// TIA Portal project "Tartak_Projekt" (V14)

(* hardware
DEVICE "S7-1200 station_1"  S7-1200 Station
   slot 0: "Rack_0"  S7-1200 Rack  Rack  V1.0
   slot 1: "PLC_1"  CPU 1214C DC/DC/DC  6ES7 214-1AG31-0XB0  V3.0
      slot 3: "AQ 1x12BIT_1"  AQ1 signal board  6ES7 232-4HA30-0XB0  V1.0
   slot 2: "DI 16/DQ 16x24VDC_1"  SM 1223 DI16/DQ16 x 24VDC  6ES7 223-1BL30-0XB0  V1.0
DEVICE "HMI_2"  TP700 Comfort
   slot 0: "TP700 Comfort"  TP700 Comfort  6AV2 124-0GC01-0AX0  14.0.1.0
   slot 1: "HMI_RT_2"  TP700 Comfort  6AV2 124-0GC01-0AX0  14.0.1.0
   slot 5: "HMI_1.IE_CP_1"  PROFINET Interface  14.0.1.0
      slot 1: "PROFINET Interface_1"  PROFINET Interface
         slot 1: "Port_1"  Port
         slot 2: "Port_2"  Port
   slot 7: "HMI_1.MPI/DP_CP_1"  MPI/DP Interface  14.0.1.0
*)

// ===== PLC "PLC_1"  CPU 1214C DC/DC/DC =====

VAR_GLOBAL   // PLC tag table "Non Default tag table2"
   "Tag_1" AT %M100.0 : Bool;
   "Tag_2" AT %M100.1 : Bool;
   "Tag_3" AT %M100.2 : Bool;
   "Tag_4" AT %M100.3 : Bool;
   "Tag_5" AT %M100.4 : Bool;
   "Tag_6" AT %M100.5 : Bool;
   "Tag_7" AT %M1000.0 : Bool;
   "Tag_8" AT %M1000.1 : Bool;
   "Tag_9" AT %M1000.2 : Bool;
   "Tag_10" AT %M1000.3 : Bool;
   "Tag_11" AT %M1000.4 : Bool;
   "Tag_12" AT %M1000.5 : Bool;
   "Tag_13" AT %M1000.6 : Bool;
   "Tag_14" AT %M1000.7 : Bool;
   "Tag_15" AT %M1001.0 : Bool;
   "Tag_16" AT %M1001.1 : Bool;
   "Tag_17" AT %M1001.2 : Bool;
   "Tag_18" AT %M1001.3 : Bool;
   "Tag_19" AT %M1002.0 : Bool;
   "Tag_20" AT %M1002.1 : Bool;
   "Tag_21" AT %M2001.0 : Bool;
END_VAR

VAR_GLOBAL   // PLC tag table "Default tag table"
   "polozenie_dluga" AT %I8.0 : Bool;
   "polozenie_srednia" AT %I8.1 : Bool;
   "polozenie_krotka" AT %I8.2 : Bool;
   "polozenie_zsyp_1" AT %I8.3 : Bool;
   "polozenie_zsyp_2" AT %I8.4 : Bool;
   "polozenie_zsyp_3" AT %I8.5 : Bool;
   "P1" AT %Q4.0 : Bool;   // Przepychacz belek krótkich
   "P2" AT %Q4.1 : Bool;   // Przepychacz belek średnich
   "P3" AT %Q4.2 : Bool;   // Przepychacz belek długich
   "otwarcie_zsyp_1" AT %Q4.3 : Bool;
   "otwarcie_zsyp_2" AT %Q4.4 : Bool;
   "otwarcie_zsyp_3" AT %Q4.5 : Bool;
   "napelnienie_zsyp_1" AT %I8.6 : Bool;
   "napelnienie_zsyp_2" AT %I8.7 : Bool;
   "napelnienie_zsyp_3" AT %I9.0 : Bool;
   "pozycja_wagnik_zsyp_1" AT %I9.7 : Bool;
   "pozycja_wagonik_zsyp_2" AT %I1.0 : Bool;
   "pozycja_wagonik_zsyp_3" AT %I1.1 : Bool;
   "ruch_wagonika" AT %Q4.6 : Bool;
   "zwrotnica_bit_0" AT %Q4.7 : Bool;
   "zwrotnica_bit_1" AT %Q5.0 : Bool;
   "bocznica_dolna_0" AT %I9.1 : Bool;
   "bocznica_dolna_1" AT %I9.2 : Bool;
   "bocznica_srodkowa_0" AT %I9.3 : Bool;
   "bocznica_srodkowa_1" AT %I9.4 : Bool;
   "bocznica_gorna_0" AT %I9.5 : Bool;
   "bocznica_gorna_1" AT %I9.6 : Bool;
   "sygnalizator_gora" AT %Q5.1 : Bool;
   "sygnalizator_srodek" AT %Q5.2 : Bool;
   "sygnalizator_dol" AT %Q5.3 : Bool;
   "Clock_Byte" AT %MB0 : Byte;
   "Clock_10Hz" AT %M0.0 : Bool;
   "Clock_5Hz" AT %M0.1 : Bool;
   "Clock_2.5Hz" AT %M0.2 : Bool;
   "Clock_2Hz" AT %M0.3 : Bool;
   "Clock_1.25Hz" AT %M0.4 : Bool;
   "Clock_1Hz" AT %M0.5 : Bool;
   "Clock_0.625Hz" AT %M0.6 : Bool;
   "Clock_0.5Hz" AT %M0.7 : Bool;
   "alarmy" AT %MW10 : Int;
   "odbiorca" AT %M12.0 : Bool;
   "zsyp_1_krotka" AT %M50.0 : Bool;
   "zsyp_1_srednia" AT %M50.1 : Bool;
   "zsyp_1_dluga" AT %M50.2 : Bool;
   "zsyp_2_krotka" AT %M50.3 : Bool;
   "zsyp_2_srednia" AT %M50.4 : Bool;
   "zsyp_2_dluga" AT %M50.5 : Bool;
   "zsyp_3_krotka" AT %M50.6 : Bool;
   "zsyp_3_srednia" AT %M50.7 : Bool;
   "zsyp_3_dluga" AT %M51.0 : Bool;
END_VAR

VAR_GLOBAL CONSTANT   // PLC tag table "Default tag table"
   "None" : Pip := 65535;
   "Automatic update" : Pip := 0;
   "PIP 1" : Pip := 1;
   "PIP 2" : Pip := 2;
   "PIP 3" : Pip := 3;
   "PIP 4" : Pip := 4;
   "PIP OB Servo" : Pip := 32768;
   "Local~MC" : Hw_SubModule := 51;
   "Local~Common" : Hw_SubModule := 50;
   "Local~Device" : Hw_Device := 32;
   "Local~Configuration" : Hw_SubModule := 33;
   "Local~Exec" : Hw_SubModule := 52;
   "Local(1)" : Hw_SubModule := 49;
   "Local~PROFINET_interface_1(1)" : Hw_Interface := 64;
   "Local~PROFINET_interface_1~Port_1(1)" : Hw_Interface := 65;
   "Local~HSC_1(1)" : Hw_Hsc := 257;
   "Local~HSC_2(1)" : Hw_Hsc := 258;
   "Local~HSC_3(1)" : Hw_Hsc := 259;
   "Local~HSC_4(1)" : Hw_Hsc := 260;
   "Local~HSC_5(1)" : Hw_Hsc := 261;
   "Local~HSC_6(1)" : Hw_Hsc := 262;
   "Local~AI_2_1(1)" : Hw_SubModule := 263;
   "Local~DI_14_DQ_10_1(1)" : Hw_SubModule := 264;
   "Local~Pulse_1(1)" : Hw_Pwm := 265;
   "Local~Pulse_2(1)" : Hw_Pwm := 266;
   "Local~Pulse_3(1)" : Hw_Pwm := 267;
   "Local~Pulse_4(1)" : Hw_Pwm := 268;
   "OB_Main(1)" : OB_PCYCLE := 1;
END_VAR

DATA_BLOCK "DB_HMI"   // DB1
{ S7_Optimized_Access := 'TRUE' }
VERSION : 0.1
   VAR
      napelnienie_zsyp_krotki : Bool;
      napelnienie_zsyp_sredni : Bool;
      napelnienie_zsyp_dlugi : Bool;
      belka_krotka : Bool;
      belka_srednia : Bool;
      belka_dluga : Bool;
      status_ruchu_wagonika : Bool;
      oproznianie_zsyp_krotki : Bool;
      oproznianie_zsyp_sredni : Bool;
      oproznianie_zsyp_dlugi : Bool;
      ustawienie_zwrotnicy : Byte;
      zapelnienie_bocznicy_krotkiej : Byte;
      zapelnienie_bocznicy_sredniej : Byte;
      zapelnienie_bocznicy_dlugiej : Byte;
      sygnalizator_bocznica_krotka : Bool;
      sygnalizator_bocznica_srednia : Bool;
      sygnalizator_bocznica_dluga : Bool;
      wagonik_krotki : Bool;
      wagonik_sredni : Bool;
      wagonik_dlugi : Bool;
      odbiorca : Bool;
      zsyp_1_krotka : Bool;
      zsyp_1_srednia : Bool;
      zsyp_1_dluga : Bool;
      zsyp_2_krotka : Bool;
      zsyp_2_srednia : Bool;
      zsyp_2_dluga : Bool;
      zsyp_3_krotka : Bool;
      zsyp_3_srednia : Bool;
      zsyp_3_dluga : Bool;
   END_VAR
BEGIN
END_DATA_BLOCK

DATA_BLOCK "wykrywanie_belki_i_zrzucanie_DB"   // DB2
{ S7_Optimized_Access := 'TRUE' }
VERSION : 0.1
// stored: InstanceOfName wykrywanie_belki_i_zrzucanie
"wykrywanie_belki_i_zrzucanie"
BEGIN
END_DATA_BLOCK

DATA_BLOCK "poruszanie_wagonikiem_i_zsypywanie_drewna_DB"   // DB3
{ S7_Optimized_Access := 'TRUE' }
VERSION : 0.1
// stored: InstanceOfName poruszanie_wagonikiem_i_zsypywanie_drewna
"poruszanie_wagonikiem_i_zsypywanie_drewna"
BEGIN
END_DATA_BLOCK

DATA_BLOCK "wykrywanie_belki_i_zrzucanie_odbiorca_DB"   // DB6
{ S7_Optimized_Access := 'TRUE' }
VERSION : 0.1
// stored: InstanceOfName wykrywanie_belki_i_zrzucanie_odbiorca
"wykrywanie_belki_i_zrzucanie_odbiorca"
BEGIN
END_DATA_BLOCK

// folder: System blocks/Program resources

DATA_BLOCK "IEC_Timer_0_DB"   // DB4
{ S7_Optimized_Access := 'TRUE' }
AUTHOR : Simatic
FAMILY : IEC
NAME : IEC_TMR
VERSION : 1.0
// stored: InstanceOfName IEC_TIMER
"IEC_TIMER"
BEGIN
END_DATA_BLOCK

DATA_BLOCK "IEC_Timer_0_DB_1"   // DB5
{ S7_Optimized_Access := 'TRUE' }
AUTHOR : Simatic
FAMILY : IEC
NAME : IEC_TMR
VERSION : 1.0
// stored: InstanceOfName IEC_TIMER
"IEC_TIMER"
BEGIN
END_DATA_BLOCK

DATA_BLOCK "IEC_Timer_0_DB_2"   // DB7
{ S7_Optimized_Access := 'TRUE' }
AUTHOR : Simatic
FAMILY : IEC
NAME : IEC_TMR
VERSION : 1.0
// stored: InstanceOfName IEC_TIMER
"IEC_TIMER"
BEGIN
END_DATA_BLOCK

// folder: (top level)

FUNCTION_BLOCK "wykrywanie_belki_i_zrzucanie"   // FB1, LAD
TITLE = Tryb normalny
{ S7_Optimized_Access := 'TRUE' }
VERSION : 0.1
// Wykrywanie belki, jej pomiar oraz zrzucanie do odpowiedniego zsypu w trybie normalnym
   VAR
      czy_wykryta_belka : Bool;
      krotka_belka : Bool;
      srednia_belka : Bool;
      dluga_belka : Bool;
      belka_zrzucona : Bool;
   END_VAR
   VAR_TEMP
      belka_na_pomiarze : Bool;
   END_VAR
   VAR_TEMP   // added for the SCL form of the ladder/FBD networks
      _w1 : Bool;
      _w2 : Bool;
      _w3 : Bool;
      _w4 : Bool;
   END_VAR
BEGIN

REGION Network 1
   // Rozpoczynanie pomiaru długości belki
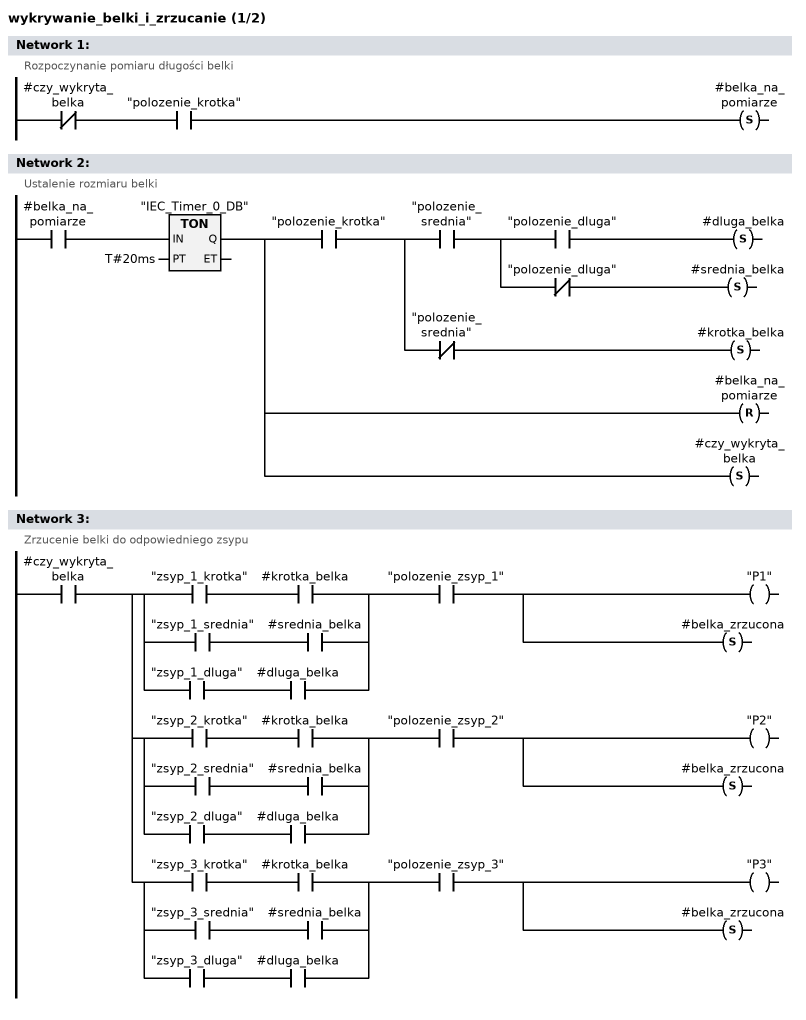
   RUNG wire#powerrail
      I_Contact( #czy_wykryta_belka )
      Contact( "polozenie_krotka" )
      S_Coil( #belka_na_pomiarze )
   END_RUNG
   // the same network as SCL:
   IF NOT #czy_wykryta_belka AND "polozenie_krotka" THEN #belka_na_pomiarze := TRUE; END_IF;
END_REGION

REGION Network 2
   // Ustalenie rozmiaru belki
   "IEC_Timer_0_DB".TON(IN := #belka_na_pomiarze, PT := T#20ms);
   #_w1 := "IEC_Timer_0_DB".Q AND "polozenie_krotka";
   #_w2 := #_w1 AND "polozenie_srednia";
   IF #_w2 AND "polozenie_dluga" THEN #dluga_belka := TRUE; END_IF;
   IF #_w2 AND NOT "polozenie_dluga" THEN #srednia_belka := TRUE; END_IF;
   IF #_w1 AND NOT "polozenie_srednia" THEN #krotka_belka := TRUE; END_IF;
   IF "IEC_Timer_0_DB".Q THEN
       #belka_na_pomiarze := FALSE;
       #czy_wykryta_belka := TRUE;
   END_IF;
END_REGION

REGION Network 3
   // Zrzucenie belki do odpowiedniego zsypu
   RUNG wire#powerrail
      Contact( #czy_wykryta_belka )
      wire#w1
      Contact( "zsyp_1_krotka" )
      Contact( #krotka_belka )
      wire#w2
      Contact( "polozenie_zsyp_1" )
      wire#w3
      Coil( "P1" )
   END_RUNG
   RUNG wire#w1
      Contact( "zsyp_1_srednia" )
      Contact( #srednia_belka )
   END_RUNG wire#w2
   RUNG wire#w1
      Contact( "zsyp_1_dluga" )
      Contact( #dluga_belka )
   END_RUNG wire#w2
   RUNG wire#w3
      S_Coil( #belka_zrzucona )
   END_RUNG
   RUNG wire#w1
      Contact( "zsyp_2_krotka" )
      Contact( #krotka_belka )
      wire#w4
      Contact( "polozenie_zsyp_2" )
      wire#w5
      Coil( "P2" )
   END_RUNG
   RUNG wire#w1
      Contact( "zsyp_2_srednia" )
      Contact( #srednia_belka )
   END_RUNG wire#w4
   RUNG wire#w1
      Contact( "zsyp_2_dluga" )
      Contact( #dluga_belka )
   END_RUNG wire#w4
   RUNG wire#w5
      S_Coil( #belka_zrzucona )
   END_RUNG
   RUNG wire#w1
      Contact( "zsyp_3_krotka" )
      Contact( #krotka_belka )
      wire#w6
      Contact( "polozenie_zsyp_3" )
      wire#w7
      Coil( "P3" )
   END_RUNG
   RUNG wire#w1
      Contact( "zsyp_3_srednia" )
      Contact( #srednia_belka )
   END_RUNG wire#w6
   RUNG wire#w1
      Contact( "zsyp_3_dluga" )
      Contact( #dluga_belka )
   END_RUNG wire#w6
   RUNG wire#w7
      S_Coil( #belka_zrzucona )
   END_RUNG
   // the same network as SCL:
   "P1" := #czy_wykryta_belka AND (("zsyp_1_krotka" AND #krotka_belka) OR ("zsyp_1_srednia" AND #srednia_belka) OR ("zsyp_1_dluga" AND #dluga_belka)) AND "polozenie_zsyp_1";
   IF "P1" THEN #belka_zrzucona := TRUE; END_IF;
   "P2" := #czy_wykryta_belka AND (("zsyp_2_krotka" AND #krotka_belka) OR ("zsyp_2_srednia" AND #srednia_belka) OR ("zsyp_2_dluga" AND #dluga_belka)) AND "polozenie_zsyp_2";
   IF "P2" THEN #belka_zrzucona := TRUE; END_IF;
   "P3" := #czy_wykryta_belka AND (("zsyp_3_krotka" AND #krotka_belka) OR ("zsyp_3_srednia" AND #srednia_belka) OR ("zsyp_3_dluga" AND #dluga_belka)) AND "polozenie_zsyp_3";
   IF "P3" THEN #belka_zrzucona := TRUE; END_IF;
END_REGION

REGION Network 4
   // Resetowanie sygnałów pomiarowych po zrzuceniu belki
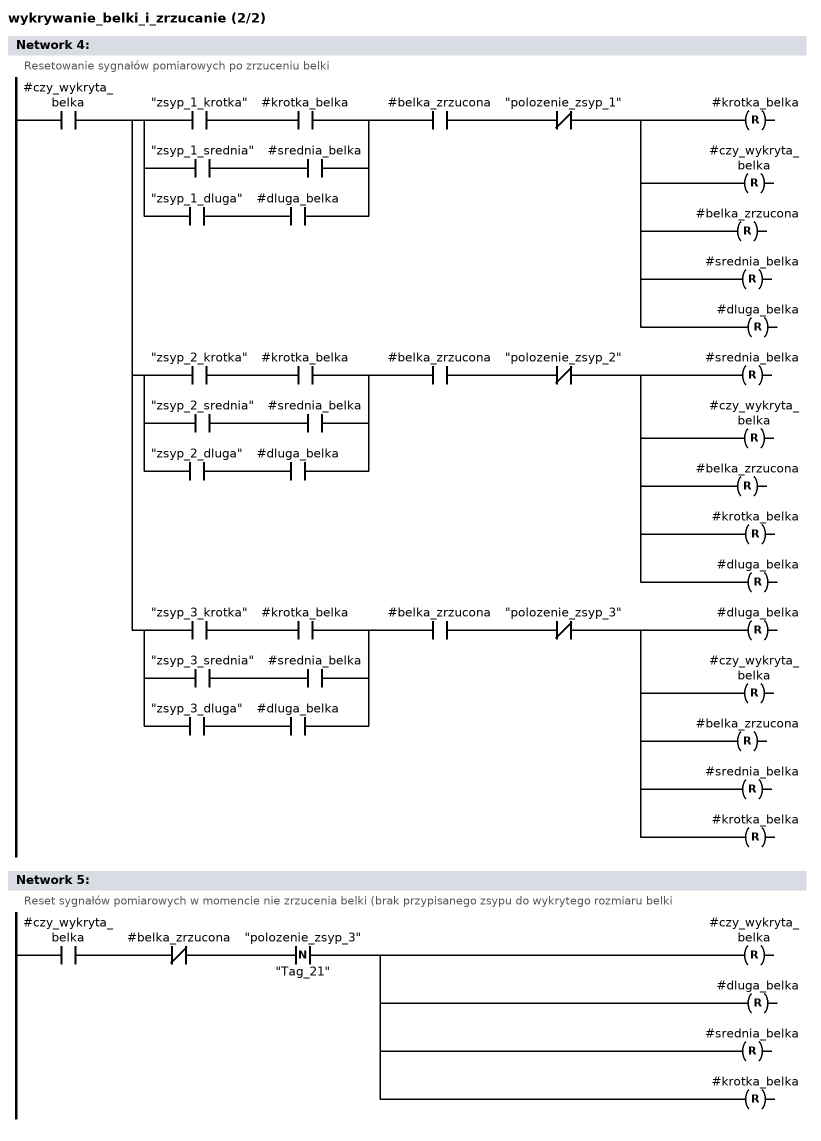
   RUNG wire#powerrail
      Contact( #czy_wykryta_belka )
      wire#w1
      Contact( "zsyp_1_krotka" )
      Contact( #krotka_belka )
      wire#w2
      Contact( #belka_zrzucona )
      I_Contact( "polozenie_zsyp_1" )
      wire#w3
      R_Coil( #krotka_belka )
   END_RUNG
   RUNG wire#w1
      Contact( "zsyp_1_srednia" )
      Contact( #srednia_belka )
   END_RUNG wire#w2
   RUNG wire#w1
      Contact( "zsyp_1_dluga" )
      Contact( #dluga_belka )
   END_RUNG wire#w2
   RUNG wire#w3
      R_Coil( #czy_wykryta_belka )
   END_RUNG
   RUNG wire#w3
      R_Coil( #belka_zrzucona )
   END_RUNG
   RUNG wire#w3
      R_Coil( #srednia_belka )
   END_RUNG
   RUNG wire#w3
      R_Coil( #dluga_belka )
   END_RUNG
   RUNG wire#w1
      Contact( "zsyp_2_krotka" )
      Contact( #krotka_belka )
      wire#w4
      Contact( #belka_zrzucona )
      I_Contact( "polozenie_zsyp_2" )
      wire#w5
      R_Coil( #srednia_belka )
   END_RUNG
   RUNG wire#w1
      Contact( "zsyp_2_srednia" )
      Contact( #srednia_belka )
   END_RUNG wire#w4
   RUNG wire#w1
      Contact( "zsyp_2_dluga" )
      Contact( #dluga_belka )
   END_RUNG wire#w4
   RUNG wire#w5
      R_Coil( #czy_wykryta_belka )
   END_RUNG
   RUNG wire#w5
      R_Coil( #belka_zrzucona )
   END_RUNG
   RUNG wire#w5
      R_Coil( #krotka_belka )
   END_RUNG
   RUNG wire#w5
      R_Coil( #dluga_belka )
   END_RUNG
   RUNG wire#w1
      Contact( "zsyp_3_krotka" )
      Contact( #krotka_belka )
      wire#w6
      Contact( #belka_zrzucona )
      I_Contact( "polozenie_zsyp_3" )
      wire#w7
      R_Coil( #dluga_belka )
   END_RUNG
   RUNG wire#w1
      Contact( "zsyp_3_srednia" )
      Contact( #srednia_belka )
   END_RUNG wire#w6
   RUNG wire#w1
      Contact( "zsyp_3_dluga" )
      Contact( #dluga_belka )
   END_RUNG wire#w6
   RUNG wire#w7
      R_Coil( #czy_wykryta_belka )
   END_RUNG
   RUNG wire#w7
      R_Coil( #belka_zrzucona )
   END_RUNG
   RUNG wire#w7
      R_Coil( #srednia_belka )
   END_RUNG
   RUNG wire#w7
      R_Coil( #krotka_belka )
   END_RUNG
   // the same network as SCL:
   #_w1 := #czy_wykryta_belka AND (("zsyp_1_krotka" AND #krotka_belka) OR ("zsyp_1_srednia" AND #srednia_belka) OR ("zsyp_1_dluga" AND #dluga_belka)) AND #belka_zrzucona AND NOT "polozenie_zsyp_1";
   IF #_w1 THEN #krotka_belka := FALSE; END_IF;
   #_w2 := #czy_wykryta_belka;
   IF #_w1 THEN
       #czy_wykryta_belka := FALSE;
       #belka_zrzucona := FALSE;
       #srednia_belka := FALSE;
       #dluga_belka := FALSE;
   END_IF;
   #_w3 := #_w2 AND (("zsyp_2_krotka" AND #krotka_belka) OR ("zsyp_2_srednia" AND #srednia_belka) OR ("zsyp_2_dluga" AND #dluga_belka)) AND #belka_zrzucona AND NOT "polozenie_zsyp_2";
   IF #_w3 THEN
       #srednia_belka := FALSE;
       #czy_wykryta_belka := FALSE;
       #belka_zrzucona := FALSE;
       #krotka_belka := FALSE;
       #dluga_belka := FALSE;
   END_IF;
   #_w4 := #_w2 AND (("zsyp_3_krotka" AND #krotka_belka) OR ("zsyp_3_srednia" AND #srednia_belka) OR ("zsyp_3_dluga" AND #dluga_belka)) AND #belka_zrzucona AND NOT "polozenie_zsyp_3";
   IF #_w4 THEN
       #dluga_belka := FALSE;
       #czy_wykryta_belka := FALSE;
       #belka_zrzucona := FALSE;
       #srednia_belka := FALSE;
       #krotka_belka := FALSE;
   END_IF;
END_REGION

REGION Network 5
   // Reset sygnałów pomiarowych w momencie nie zrzucenia belki (brak przypisanego zsypu do wykrytego rozmiaru belki
   RUNG wire#powerrail
      Contact( #czy_wykryta_belka )
      I_Contact( #belka_zrzucona )
      N_Contact(operand := "polozenie_zsyp_3", bit := "Tag_21")
      wire#w1
      R_Coil( #czy_wykryta_belka )
   END_RUNG
   RUNG wire#w1
      R_Coil( #dluga_belka )
   END_RUNG
   RUNG wire#w1
      R_Coil( #srednia_belka )
   END_RUNG
   RUNG wire#w1
      R_Coil( #krotka_belka )
   END_RUNG
   // the same network as SCL:
   #_w1 := #czy_wykryta_belka AND NOT #belka_zrzucona AND NOT "polozenie_zsyp_3" AND "Tag_21";   // falling edge of "polozenie_zsyp_3"
   "Tag_21" := "polozenie_zsyp_3";
   IF #_w1 THEN
       #czy_wykryta_belka := FALSE;
       #dluga_belka := FALSE;
       #srednia_belka := FALSE;
       #krotka_belka := FALSE;
   END_IF;
END_REGION
END_FUNCTION_BLOCK

FUNCTION_BLOCK "poruszanie_wagonikiem_i_zsypywanie_drewna"   // FB2, LAD
{ S7_Optimized_Access := 'TRUE' }
VERSION : 0.1
// Opróżnianie zsypów, ustawianie wagoników na odpowiedniej bocznicy oraz opuszczanie tartaku
   VAR
      wagonik_krotki : Bool;
      wagonik_sredni : Bool;
      wagonik_dlugi : Bool;
   END_VAR
   VAR_TEMP   // added for the SCL form of the ladder/FBD networks
      _w1 : Bool;
      _w2 : Bool;
      _w3 : Bool;
      _w4 : Bool;
      _w5 : Bool;
      _w6 : Bool;
   END_VAR
BEGIN

REGION Network 1
   // Poruszanie wagonika w momencie napełnienia zsypu
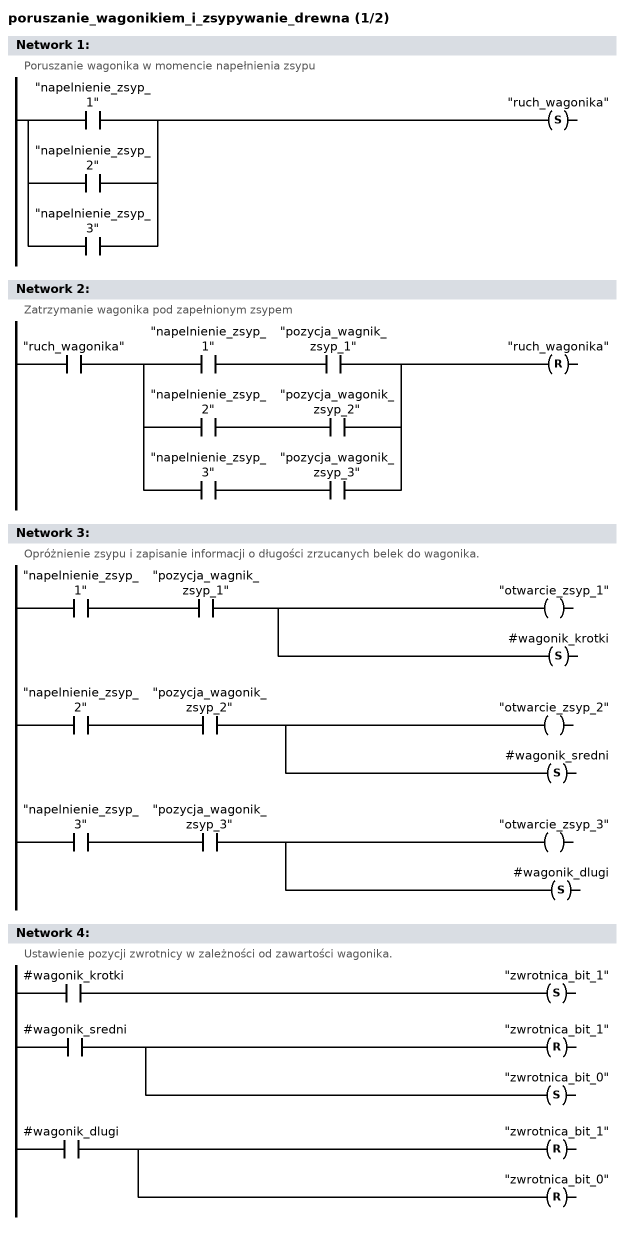
   RUNG wire#powerrail
      Contact( "napelnienie_zsyp_1" )
      wire#w1
      S_Coil( "ruch_wagonika" )
   END_RUNG
   RUNG wire#powerrail
      Contact( "napelnienie_zsyp_2" )
   END_RUNG wire#w1
   RUNG wire#powerrail
      Contact( "napelnienie_zsyp_3" )
   END_RUNG wire#w1
   // the same network as SCL:
   IF "napelnienie_zsyp_1" OR "napelnienie_zsyp_2" OR "napelnienie_zsyp_3" THEN
       "ruch_wagonika" := TRUE;
   END_IF;
END_REGION

REGION Network 2
   // Zatrzymanie wagonika pod zapełnionym zsypem
   RUNG wire#powerrail
      Contact( "ruch_wagonika" )
      wire#w1
      Contact( "napelnienie_zsyp_1" )
      Contact( "pozycja_wagnik_zsyp_1" )
      wire#w2
      R_Coil( "ruch_wagonika" )
   END_RUNG
   RUNG wire#w1
      Contact( "napelnienie_zsyp_2" )
      Contact( "pozycja_wagonik_zsyp_2" )
   END_RUNG wire#w2
   RUNG wire#w1
      Contact( "napelnienie_zsyp_3" )
      Contact( "pozycja_wagonik_zsyp_3" )
   END_RUNG wire#w2
   // the same network as SCL:
   IF "ruch_wagonika" AND (("napelnienie_zsyp_1" AND "pozycja_wagnik_zsyp_1") OR ("napelnienie_zsyp_2" AND "pozycja_wagonik_zsyp_2") OR ("napelnienie_zsyp_3" AND "pozycja_wagonik_zsyp_3")) THEN
       "ruch_wagonika" := FALSE;
   END_IF;
END_REGION

REGION Network 3
   // Opróżnienie zsypu i zapisanie informacji o długości zrzucanych belek do wagonika.
   RUNG wire#powerrail
      Contact( "napelnienie_zsyp_1" )
      Contact( "pozycja_wagnik_zsyp_1" )
      wire#w1
      Coil( "otwarcie_zsyp_1" )
   END_RUNG
   RUNG wire#w1
      S_Coil( #wagonik_krotki )
   END_RUNG
   RUNG wire#powerrail
      Contact( "napelnienie_zsyp_2" )
      Contact( "pozycja_wagonik_zsyp_2" )
      wire#w2
      Coil( "otwarcie_zsyp_2" )
   END_RUNG
   RUNG wire#w2
      S_Coil( #wagonik_sredni )
   END_RUNG
   RUNG wire#powerrail
      Contact( "napelnienie_zsyp_3" )
      Contact( "pozycja_wagonik_zsyp_3" )
      wire#w3
      Coil( "otwarcie_zsyp_3" )
   END_RUNG
   RUNG wire#w3
      S_Coil( #wagonik_dlugi )
   END_RUNG
   // the same network as SCL:
   "otwarcie_zsyp_1" := "napelnienie_zsyp_1" AND "pozycja_wagnik_zsyp_1";
   IF "otwarcie_zsyp_1" THEN #wagonik_krotki := TRUE; END_IF;
   "otwarcie_zsyp_2" := "napelnienie_zsyp_2" AND "pozycja_wagonik_zsyp_2";
   IF "otwarcie_zsyp_2" THEN #wagonik_sredni := TRUE; END_IF;
   "otwarcie_zsyp_3" := "napelnienie_zsyp_3" AND "pozycja_wagonik_zsyp_3";
   IF "otwarcie_zsyp_3" THEN #wagonik_dlugi := TRUE; END_IF;
END_REGION

REGION Network 4
   // Ustawienie pozycji zwrotnicy w zależności od zawartości wagonika.
   RUNG wire#powerrail
      Contact( #wagonik_krotki )
      S_Coil( "zwrotnica_bit_1" )
   END_RUNG
   RUNG wire#powerrail
      Contact( #wagonik_sredni )
      wire#w1
      R_Coil( "zwrotnica_bit_1" )
   END_RUNG
   RUNG wire#w1
      S_Coil( "zwrotnica_bit_0" )
   END_RUNG
   RUNG wire#powerrail
      Contact( #wagonik_dlugi )
      wire#w2
      R_Coil( "zwrotnica_bit_1" )
   END_RUNG
   RUNG wire#w2
      R_Coil( "zwrotnica_bit_0" )
   END_RUNG
   // the same network as SCL:
   IF #wagonik_krotki THEN "zwrotnica_bit_1" := TRUE; END_IF;
   IF #wagonik_sredni THEN
       "zwrotnica_bit_1" := FALSE;
       "zwrotnica_bit_0" := TRUE;
   END_IF;
   IF #wagonik_dlugi THEN
       "zwrotnica_bit_1" := FALSE;
       "zwrotnica_bit_0" := FALSE;
   END_IF;
END_REGION

REGION Network 5
   // Przejazd wagonika na bocznicę.
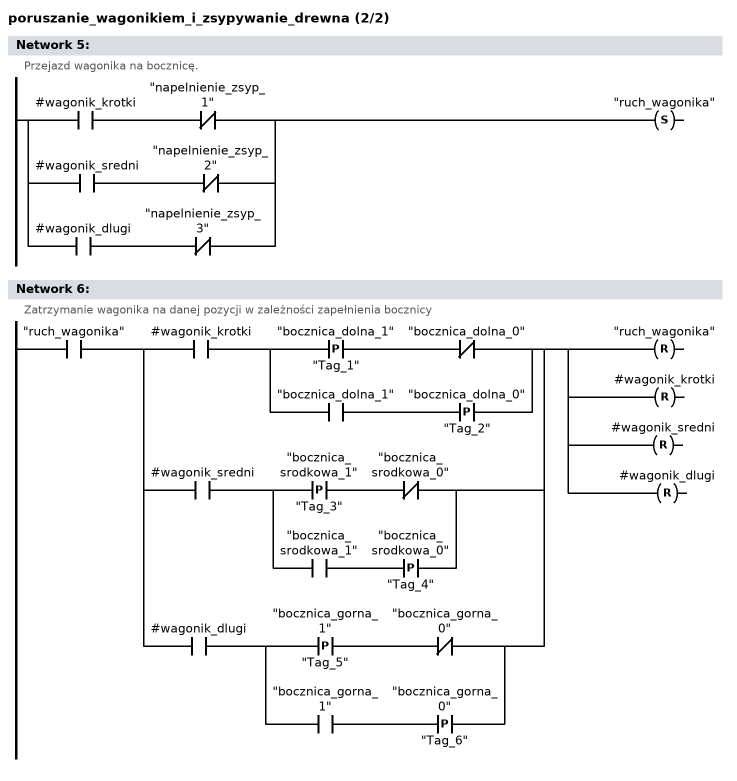
   RUNG wire#powerrail
      Contact( #wagonik_krotki )
      I_Contact( "napelnienie_zsyp_1" )
      wire#w1
      S_Coil( "ruch_wagonika" )
   END_RUNG
   RUNG wire#powerrail
      Contact( #wagonik_sredni )
      I_Contact( "napelnienie_zsyp_2" )
   END_RUNG wire#w1
   RUNG wire#powerrail
      Contact( #wagonik_dlugi )
      I_Contact( "napelnienie_zsyp_3" )
   END_RUNG wire#w1
   // the same network as SCL:
   IF (#wagonik_krotki AND NOT "napelnienie_zsyp_1") OR (#wagonik_sredni AND NOT "napelnienie_zsyp_2") OR (#wagonik_dlugi AND NOT "napelnienie_zsyp_3") THEN
       "ruch_wagonika" := TRUE;
   END_IF;
END_REGION

REGION Network 6
   // Zatrzymanie wagonika na danej pozycji w zależności zapełnienia bocznicy
   RUNG wire#powerrail
      Contact( "ruch_wagonika" )
      wire#w1
      Contact( #wagonik_krotki )
      wire#w2
      P_Contact(operand := "bocznica_dolna_1", bit := "Tag_1")
      I_Contact( "bocznica_dolna_0" )
      wire#w3
      R_Coil( "ruch_wagonika" )
   END_RUNG
   RUNG wire#w2
      Contact( "bocznica_dolna_1" )
      P_Contact(operand := "bocznica_dolna_0", bit := "Tag_2")
   END_RUNG wire#w3
   RUNG wire#w1
      Contact( #wagonik_sredni )
      wire#w4
      P_Contact(operand := "bocznica_srodkowa_1", bit := "Tag_3")
      I_Contact( "bocznica_srodkowa_0" )
   END_RUNG wire#w3
   RUNG wire#w4
      Contact( "bocznica_srodkowa_1" )
      P_Contact(operand := "bocznica_srodkowa_0", bit := "Tag_4")
   END_RUNG wire#w3
   RUNG wire#w1
      Contact( #wagonik_dlugi )
      wire#w5
      P_Contact(operand := "bocznica_gorna_1", bit := "Tag_5")
      I_Contact( "bocznica_gorna_0" )
   END_RUNG wire#w3
   RUNG wire#w5
      Contact( "bocznica_gorna_1" )
      P_Contact(operand := "bocznica_gorna_0", bit := "Tag_6")
   END_RUNG wire#w3
   RUNG wire#w3
      R_Coil( #wagonik_krotki )
   END_RUNG
   RUNG wire#w3
      R_Coil( #wagonik_sredni )
   END_RUNG
   RUNG wire#w3
      R_Coil( #wagonik_dlugi )
   END_RUNG
   // the same network as SCL:
   #_w1 := "ruch_wagonika" AND #wagonik_krotki AND "bocznica_dolna_1" AND NOT "Tag_1";   // rising edge of "bocznica_dolna_1"
   "Tag_1" := "bocznica_dolna_1";
   #_w2 := "ruch_wagonika" AND #wagonik_krotki AND "bocznica_dolna_1" AND "bocznica_dolna_0" AND NOT "Tag_2";   // rising edge of "bocznica_dolna_0"
   "Tag_2" := "bocznica_dolna_0";
   #_w3 := "ruch_wagonika" AND #wagonik_sredni AND "bocznica_srodkowa_1" AND NOT "Tag_3";   // rising edge of "bocznica_srodkowa_1"
   "Tag_3" := "bocznica_srodkowa_1";
   #_w4 := "ruch_wagonika" AND #wagonik_sredni AND "bocznica_srodkowa_1" AND "bocznica_srodkowa_0" AND NOT "Tag_4";   // rising edge of "bocznica_srodkowa_0"
   "Tag_4" := "bocznica_srodkowa_0";
   #_w5 := "ruch_wagonika" AND #wagonik_dlugi AND "bocznica_gorna_1" AND NOT "Tag_5";   // rising edge of "bocznica_gorna_1"
   "Tag_5" := "bocznica_gorna_1";
   #_w6 := "ruch_wagonika" AND #wagonik_dlugi AND "bocznica_gorna_1" AND "bocznica_gorna_0" AND NOT "Tag_6";   // rising edge of "bocznica_gorna_0"
   "Tag_6" := "bocznica_gorna_0";
   IF (#_w1 AND NOT "bocznica_dolna_0") OR #_w2 OR (#_w3 AND NOT "bocznica_srodkowa_0") OR #_w4 OR (#_w5 AND NOT "bocznica_gorna_0") OR #_w6 THEN
       "ruch_wagonika" := FALSE;
       #wagonik_krotki := FALSE;
       #wagonik_sredni := FALSE;
       #wagonik_dlugi := FALSE;
   END_IF;
END_REGION
END_FUNCTION_BLOCK

FUNCTION_BLOCK "wykrywanie_belki_i_zrzucanie_odbiorca"   // FB3, LAD
TITLE = Tryb uniwersalnego odbiorcy
{ S7_Optimized_Access := 'TRUE' }
VERSION : 0.1
// Wykrywanie belki, jej pomiar oraz zrzucanie do odpowiedniego zsypu w trybie uniwersalnego odbiorcy
   VAR
      czy_wykryta_belka : Bool;
      belka_zrzucona : Bool;
      krotka_belka : Bool;
      srednia_belka : Bool;
      dluga_belka : Bool;
   END_VAR
   VAR_TEMP
      belka_na_pomiarze : Bool;
   END_VAR
   VAR_TEMP   // added for the SCL form of the ladder/FBD networks
      _w1 : Bool;
      _w2 : Bool;
   END_VAR
BEGIN

REGION Network 1
   // Rozpoczynanie pomiaru długości belki
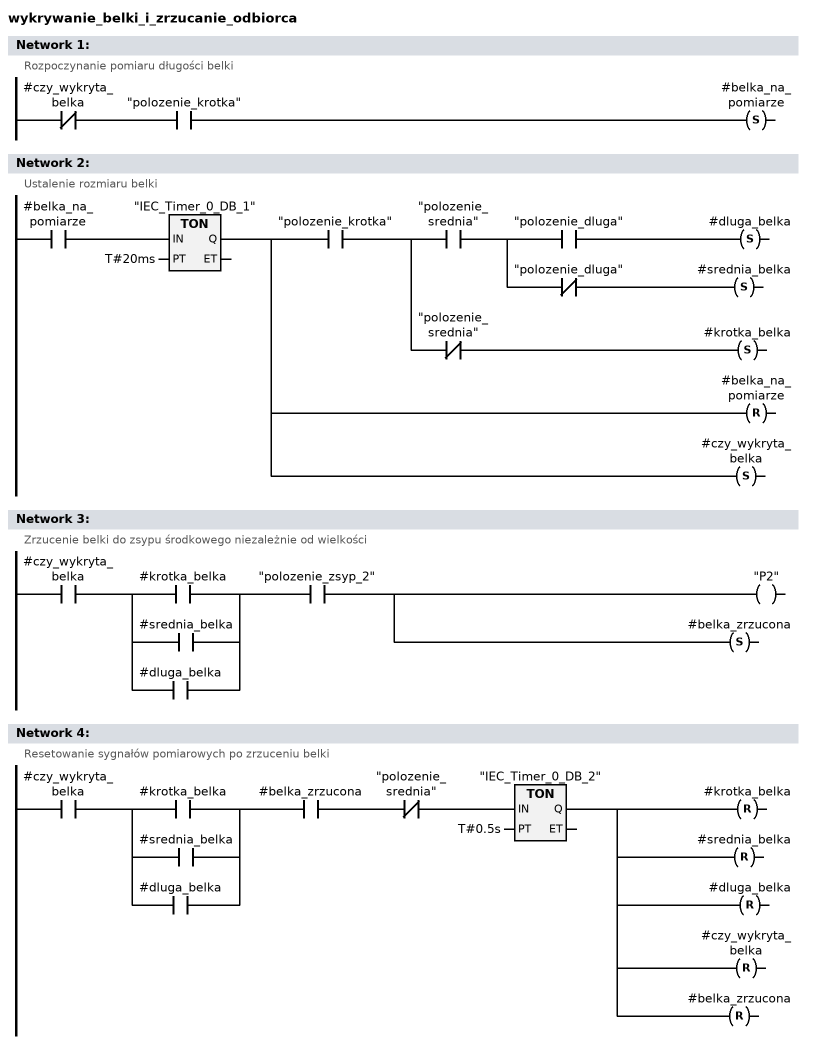
   RUNG wire#powerrail
      I_Contact( #czy_wykryta_belka )
      Contact( "polozenie_krotka" )
      S_Coil( #belka_na_pomiarze )
   END_RUNG
   // the same network as SCL:
   IF NOT #czy_wykryta_belka AND "polozenie_krotka" THEN #belka_na_pomiarze := TRUE; END_IF;
END_REGION

REGION Network 2
   // Ustalenie rozmiaru belki
   "IEC_Timer_0_DB_1".TON(IN := #belka_na_pomiarze, PT := T#20ms);
   #_w1 := "IEC_Timer_0_DB_1".Q AND "polozenie_krotka";
   #_w2 := #_w1 AND "polozenie_srednia";
   IF #_w2 AND "polozenie_dluga" THEN #dluga_belka := TRUE; END_IF;
   IF #_w2 AND NOT "polozenie_dluga" THEN #srednia_belka := TRUE; END_IF;
   IF #_w1 AND NOT "polozenie_srednia" THEN #krotka_belka := TRUE; END_IF;
   IF "IEC_Timer_0_DB_1".Q THEN
       #belka_na_pomiarze := FALSE;
       #czy_wykryta_belka := TRUE;
   END_IF;
END_REGION

REGION Network 3
   // Zrzucenie belki do zsypu środkowego niezależnie od wielkości
   RUNG wire#powerrail
      Contact( #czy_wykryta_belka )
      wire#w1
      Contact( #krotka_belka )
      wire#w2
      Contact( "polozenie_zsyp_2" )
      wire#w3
      Coil( "P2" )
   END_RUNG
   RUNG wire#w1
      Contact( #srednia_belka )
   END_RUNG wire#w2
   RUNG wire#w1
      Contact( #dluga_belka )
   END_RUNG wire#w2
   RUNG wire#w3
      S_Coil( #belka_zrzucona )
   END_RUNG
   // the same network as SCL:
   "P2" := #czy_wykryta_belka AND (#krotka_belka OR #srednia_belka OR #dluga_belka) AND "polozenie_zsyp_2";
   IF "P2" THEN #belka_zrzucona := TRUE; END_IF;
END_REGION

REGION Network 4
   // Resetowanie sygnałów pomiarowych po zrzuceniu belki
   "IEC_Timer_0_DB_2".TON(IN := #czy_wykryta_belka AND (#krotka_belka OR #srednia_belka OR #dluga_belka) AND #belka_zrzucona AND NOT "polozenie_srednia",
                          PT := T#0.5s);
   IF "IEC_Timer_0_DB_2".Q THEN
       #krotka_belka := FALSE;
       #srednia_belka := FALSE;
       #dluga_belka := FALSE;
       #czy_wykryta_belka := FALSE;
       #belka_zrzucona := FALSE;
   END_IF;
END_REGION
END_FUNCTION_BLOCK

FUNCTION "przepisywanie_HMI" : Void   // FC1, LAD
{ S7_Optimized_Access := 'TRUE' }
VERSION : 0.1
   VAR_TEMP   // added for the SCL form of the ladder/FBD networks
      _w1 : Bool;
      _w2 : Bool;
      _w3 : Bool;
      _w4 : Bool;
      _w5 : Bool;
      _w6 : Bool;
   END_VAR
BEGIN

REGION Network 1: Wykryte rozmiary belek
   // Ustawianie rozmiaru belki
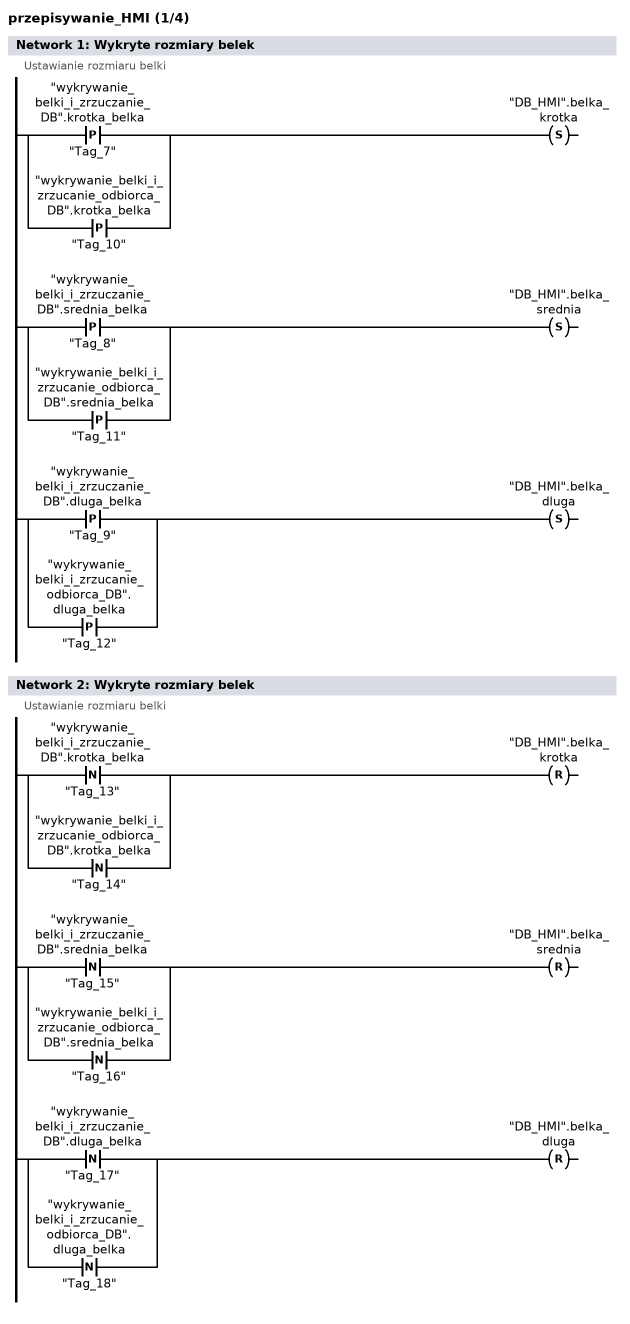
   RUNG wire#powerrail
      P_Contact(operand := "wykrywanie_belki_i_zrzuczanie_DB".krotka_belka, bit := "Tag_7")
      wire#w1
      S_Coil( "DB_HMI".belka_krotka )
   END_RUNG
   RUNG wire#powerrail
      P_Contact(operand := "wykrywanie_belki_i_zrzucanie_odbiorca_DB".krotka_belka, bit := "Tag_10")
   END_RUNG wire#w1
   RUNG wire#powerrail
      P_Contact(operand := "wykrywanie_belki_i_zrzuczanie_DB".srednia_belka, bit := "Tag_8")
      wire#w2
      S_Coil( "DB_HMI".belka_srednia )
   END_RUNG
   RUNG wire#powerrail
      P_Contact(operand := "wykrywanie_belki_i_zrzucanie_odbiorca_DB".srednia_belka, bit := "Tag_11")
   END_RUNG wire#w2
   RUNG wire#powerrail
      P_Contact(operand := "wykrywanie_belki_i_zrzuczanie_DB".dluga_belka, bit := "Tag_9")
      wire#w3
      S_Coil( "DB_HMI".belka_dluga )
   END_RUNG
   RUNG wire#powerrail
      P_Contact(operand := "wykrywanie_belki_i_zrzucanie_odbiorca_DB".dluga_belka, bit := "Tag_12")
   END_RUNG wire#w3
   // the same network as SCL:
   #_w1 := "wykrywanie_belki_i_zrzuczanie_DB".krotka_belka AND NOT "Tag_7";   // rising edge of "wykrywanie_belki_i_zrzuczanie_DB".krotka_belka
   "Tag_7" := "wykrywanie_belki_i_zrzuczanie_DB".krotka_belka;
   #_w2 := "wykrywanie_belki_i_zrzucanie_odbiorca_DB".krotka_belka AND NOT "Tag_10";   // rising edge of "wykrywanie_belki_i_zrzucanie_odbiorca_DB".krotka_belka
   "Tag_10" := "wykrywanie_belki_i_zrzucanie_odbiorca_DB".krotka_belka;
   IF #_w1 OR #_w2 THEN "DB_HMI".belka_krotka := TRUE; END_IF;
   #_w3 := "wykrywanie_belki_i_zrzuczanie_DB".srednia_belka AND NOT "Tag_8";   // rising edge of "wykrywanie_belki_i_zrzuczanie_DB".srednia_belka
   "Tag_8" := "wykrywanie_belki_i_zrzuczanie_DB".srednia_belka;
   #_w4 := "wykrywanie_belki_i_zrzucanie_odbiorca_DB".srednia_belka AND NOT "Tag_11";   // rising edge of "wykrywanie_belki_i_zrzucanie_odbiorca_DB".srednia_belka
   "Tag_11" := "wykrywanie_belki_i_zrzucanie_odbiorca_DB".srednia_belka;
   IF #_w3 OR #_w4 THEN "DB_HMI".belka_srednia := TRUE; END_IF;
   #_w5 := "wykrywanie_belki_i_zrzuczanie_DB".dluga_belka AND NOT "Tag_9";   // rising edge of "wykrywanie_belki_i_zrzuczanie_DB".dluga_belka
   "Tag_9" := "wykrywanie_belki_i_zrzuczanie_DB".dluga_belka;
   #_w6 := "wykrywanie_belki_i_zrzucanie_odbiorca_DB".dluga_belka AND NOT "Tag_12";   // rising edge of "wykrywanie_belki_i_zrzucanie_odbiorca_DB".dluga_belka
   "Tag_12" := "wykrywanie_belki_i_zrzucanie_odbiorca_DB".dluga_belka;
   IF #_w5 OR #_w6 THEN "DB_HMI".belka_dluga := TRUE; END_IF;
END_REGION

REGION Network 2: Wykryte rozmiary belek
   // Ustawianie rozmiaru belki
   RUNG wire#powerrail
      N_Contact(operand := "wykrywanie_belki_i_zrzuczanie_DB".krotka_belka, bit := "Tag_13")
      wire#w1
      R_Coil( "DB_HMI".belka_krotka )
   END_RUNG
   RUNG wire#powerrail
      N_Contact(operand := "wykrywanie_belki_i_zrzucanie_odbiorca_DB".krotka_belka, bit := "Tag_14")
   END_RUNG wire#w1
   RUNG wire#powerrail
      N_Contact(operand := "wykrywanie_belki_i_zrzuczanie_DB".srednia_belka, bit := "Tag_15")
      wire#w2
      R_Coil( "DB_HMI".belka_srednia )
   END_RUNG
   RUNG wire#powerrail
      N_Contact(operand := "wykrywanie_belki_i_zrzucanie_odbiorca_DB".srednia_belka, bit := "Tag_16")
   END_RUNG wire#w2
   RUNG wire#powerrail
      N_Contact(operand := "wykrywanie_belki_i_zrzuczanie_DB".dluga_belka, bit := "Tag_17")
      wire#w3
      R_Coil( "DB_HMI".belka_dluga )
   END_RUNG
   RUNG wire#powerrail
      N_Contact(operand := "wykrywanie_belki_i_zrzucanie_odbiorca_DB".dluga_belka, bit := "Tag_18")
   END_RUNG wire#w3
   // the same network as SCL:
   #_w1 := NOT "wykrywanie_belki_i_zrzuczanie_DB".krotka_belka AND "Tag_13";   // falling edge of "wykrywanie_belki_i_zrzuczanie_DB".krotka_belka
   "Tag_13" := "wykrywanie_belki_i_zrzuczanie_DB".krotka_belka;
   #_w2 := NOT "wykrywanie_belki_i_zrzucanie_odbiorca_DB".krotka_belka AND "Tag_14";   // falling edge of "wykrywanie_belki_i_zrzucanie_odbiorca_DB".krotka_belka
   "Tag_14" := "wykrywanie_belki_i_zrzucanie_odbiorca_DB".krotka_belka;
   IF #_w1 OR #_w2 THEN "DB_HMI".belka_krotka := FALSE; END_IF;
   #_w3 := NOT "wykrywanie_belki_i_zrzuczanie_DB".srednia_belka AND "Tag_15";   // falling edge of "wykrywanie_belki_i_zrzuczanie_DB".srednia_belka
   "Tag_15" := "wykrywanie_belki_i_zrzuczanie_DB".srednia_belka;
   #_w4 := NOT "wykrywanie_belki_i_zrzucanie_odbiorca_DB".srednia_belka AND "Tag_16";   // falling edge of "wykrywanie_belki_i_zrzucanie_odbiorca_DB".srednia_belka
   "Tag_16" := "wykrywanie_belki_i_zrzucanie_odbiorca_DB".srednia_belka;
   IF #_w3 OR #_w4 THEN "DB_HMI".belka_srednia := FALSE; END_IF;
   #_w5 := NOT "wykrywanie_belki_i_zrzuczanie_DB".dluga_belka AND "Tag_17";   // falling edge of "wykrywanie_belki_i_zrzuczanie_DB".dluga_belka
   "Tag_17" := "wykrywanie_belki_i_zrzuczanie_DB".dluga_belka;
   #_w6 := NOT "wykrywanie_belki_i_zrzucanie_odbiorca_DB".dluga_belka AND "Tag_18";   // falling edge of "wykrywanie_belki_i_zrzucanie_odbiorca_DB".dluga_belka
   "Tag_18" := "wykrywanie_belki_i_zrzucanie_odbiorca_DB".dluga_belka;
   IF #_w5 OR #_w6 THEN "DB_HMI".belka_dluga := FALSE; END_IF;
END_REGION

REGION Network 3: Napełnianie zsypów
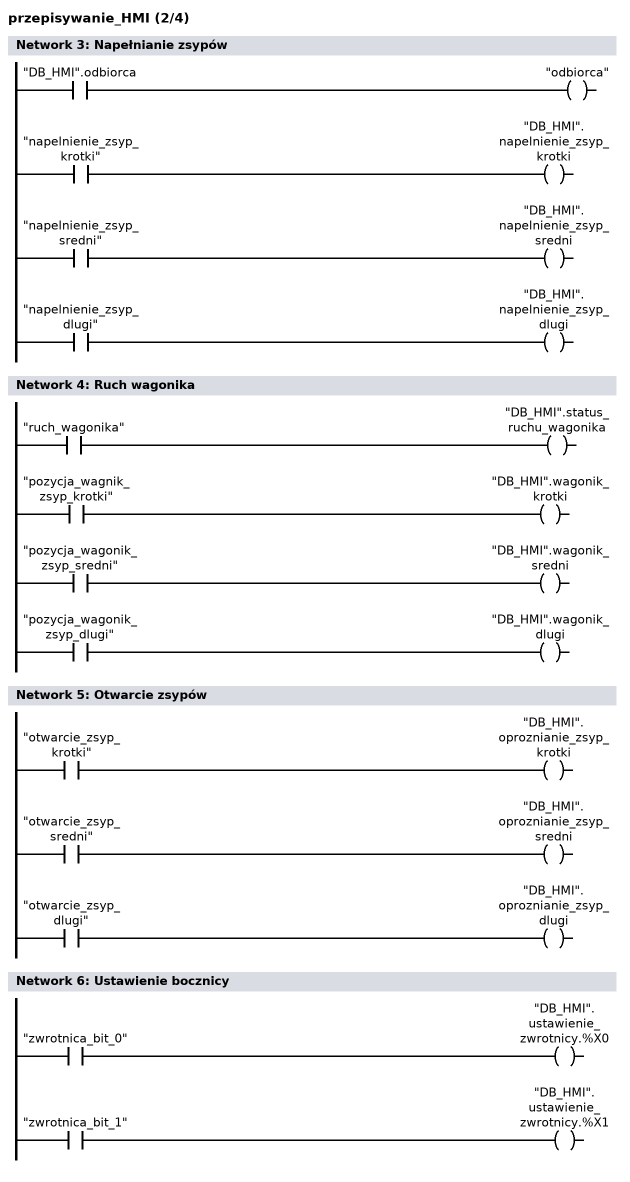
   RUNG wire#powerrail
      Contact( "DB_HMI".odbiorca )
      Coil( "odbiorca" )
   END_RUNG
   RUNG wire#powerrail
      Contact( "napelnienie_zsyp_krotki" )
      Coil( "DB_HMI".napelnienie_zsyp_krotki )
   END_RUNG
   RUNG wire#powerrail
      Contact( "napelnienie_zsyp_sredni" )
      Coil( "DB_HMI".napelnienie_zsyp_sredni )
   END_RUNG
   RUNG wire#powerrail
      Contact( "napelnienie_zsyp_dlugi" )
      Coil( "DB_HMI".napelnienie_zsyp_dlugi )
   END_RUNG
   // the same network as SCL:
   "odbiorca" := "DB_HMI".odbiorca;
   "DB_HMI".napelnienie_zsyp_krotki := "napelnienie_zsyp_krotki";
   "DB_HMI".napelnienie_zsyp_sredni := "napelnienie_zsyp_sredni";
   "DB_HMI".napelnienie_zsyp_dlugi := "napelnienie_zsyp_dlugi";
END_REGION

REGION Network 4: Ruch wagonika
   RUNG wire#powerrail
      Contact( "ruch_wagonika" )
      Coil( "DB_HMI".status_ruchu_wagonika )
   END_RUNG
   RUNG wire#powerrail
      Contact( "pozycja_wagnik_zsyp_krotki" )
      Coil( "DB_HMI".wagonik_krotki )
   END_RUNG
   RUNG wire#powerrail
      Contact( "pozycja_wagonik_zsyp_sredni" )
      Coil( "DB_HMI".wagonik_sredni )
   END_RUNG
   RUNG wire#powerrail
      Contact( "pozycja_wagonik_zsyp_dlugi" )
      Coil( "DB_HMI".wagonik_dlugi )
   END_RUNG
   // the same network as SCL:
   "DB_HMI".status_ruchu_wagonika := "ruch_wagonika";
   "DB_HMI".wagonik_krotki := "pozycja_wagnik_zsyp_krotki";
   "DB_HMI".wagonik_sredni := "pozycja_wagonik_zsyp_sredni";
   "DB_HMI".wagonik_dlugi := "pozycja_wagonik_zsyp_dlugi";
END_REGION

REGION Network 5: Otwarcie zsypów
   RUNG wire#powerrail
      Contact( "otwarcie_zsyp_krotki" )
      Coil( "DB_HMI".oproznianie_zsyp_krotki )
   END_RUNG
   RUNG wire#powerrail
      Contact( "otwarcie_zsyp_sredni" )
      Coil( "DB_HMI".oproznianie_zsyp_sredni )
   END_RUNG
   RUNG wire#powerrail
      Contact( "otwarcie_zsyp_dlugi" )
      Coil( "DB_HMI".oproznianie_zsyp_dlugi )
   END_RUNG
   // the same network as SCL:
   "DB_HMI".oproznianie_zsyp_krotki := "otwarcie_zsyp_krotki";
   "DB_HMI".oproznianie_zsyp_sredni := "otwarcie_zsyp_sredni";
   "DB_HMI".oproznianie_zsyp_dlugi := "otwarcie_zsyp_dlugi";
END_REGION

REGION Network 6: Ustawienie bocznicy
   RUNG wire#powerrail
      Contact( "zwrotnica_bit_0" )
      Coil( "DB_HMI".ustawienie_zwrotnicy.%X0 )
   END_RUNG
   RUNG wire#powerrail
      Contact( "zwrotnica_bit_1" )
      Coil( "DB_HMI".ustawienie_zwrotnicy.%X1 )
   END_RUNG
   // the same network as SCL:
   "DB_HMI".ustawienie_zwrotnicy.%X0 := "zwrotnica_bit_0";
   "DB_HMI".ustawienie_zwrotnicy.%X1 := "zwrotnica_bit_1";
END_REGION

REGION Network 7: Zapełnienie bocznic
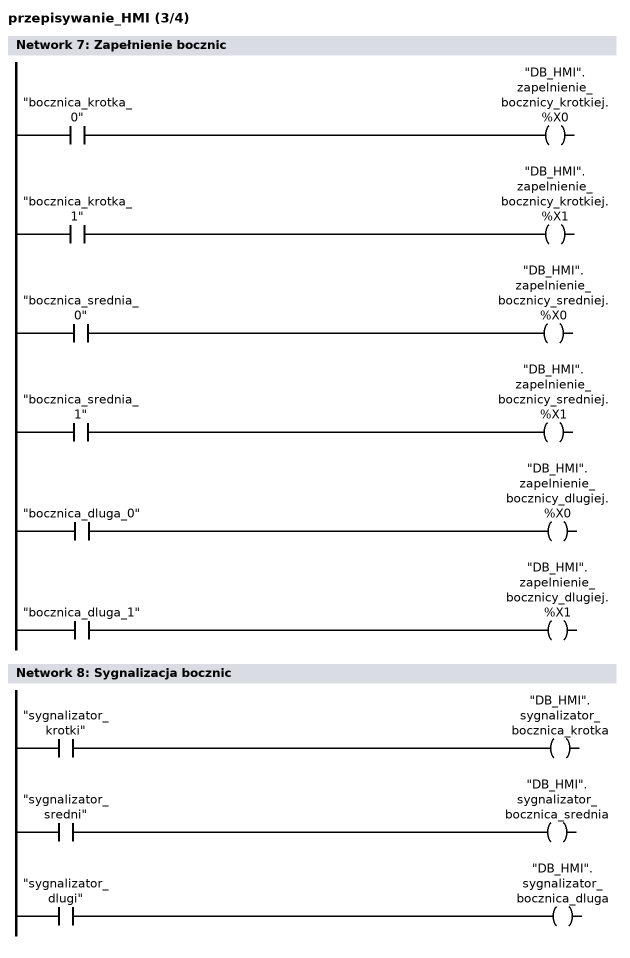
   RUNG wire#powerrail
      Contact( "bocznica_krotka_0" )
      Coil( "DB_HMI".zapelnienie_bocznicy_krotkiej.%X0 )
   END_RUNG
   RUNG wire#powerrail
      Contact( "bocznica_krotka_1" )
      Coil( "DB_HMI".zapelnienie_bocznicy_krotkiej.%X1 )
   END_RUNG
   RUNG wire#powerrail
      Contact( "bocznica_srednia_0" )
      Coil( "DB_HMI".zapelnienie_bocznicy_sredniej.%X0 )
   END_RUNG
   RUNG wire#powerrail
      Contact( "bocznica_srednia_1" )
      Coil( "DB_HMI".zapelnienie_bocznicy_sredniej.%X1 )
   END_RUNG
   RUNG wire#powerrail
      Contact( "bocznica_dluga_0" )
      Coil( "DB_HMI".zapelnienie_bocznicy_dlugiej.%X0 )
   END_RUNG
   RUNG wire#powerrail
      Contact( "bocznica_dluga_1" )
      Coil( "DB_HMI".zapelnienie_bocznicy_dlugiej.%X1 )
   END_RUNG
   // the same network as SCL:
   "DB_HMI".zapelnienie_bocznicy_krotkiej.%X0 := "bocznica_krotka_0";
   "DB_HMI".zapelnienie_bocznicy_krotkiej.%X1 := "bocznica_krotka_1";
   "DB_HMI".zapelnienie_bocznicy_sredniej.%X0 := "bocznica_srednia_0";
   "DB_HMI".zapelnienie_bocznicy_sredniej.%X1 := "bocznica_srednia_1";
   "DB_HMI".zapelnienie_bocznicy_dlugiej.%X0 := "bocznica_dluga_0";
   "DB_HMI".zapelnienie_bocznicy_dlugiej.%X1 := "bocznica_dluga_1";
END_REGION

REGION Network 8: Sygnalizacja bocznic
   RUNG wire#powerrail
      Contact( "sygnalizator_krotki" )
      Coil( "DB_HMI".sygnalizator_bocznica_krotka )
   END_RUNG
   RUNG wire#powerrail
      Contact( "sygnalizator_sredni" )
      Coil( "DB_HMI".sygnalizator_bocznica_srednia )
   END_RUNG
   RUNG wire#powerrail
      Contact( "sygnalizator_dlugi" )
      Coil( "DB_HMI".sygnalizator_bocznica_dluga )
   END_RUNG
   // the same network as SCL:
   "DB_HMI".sygnalizator_bocznica_krotka := "sygnalizator_krotki";
   "DB_HMI".sygnalizator_bocznica_srednia := "sygnalizator_sredni";
   "DB_HMI".sygnalizator_bocznica_dluga := "sygnalizator_dlugi";
END_REGION

REGION Network 9
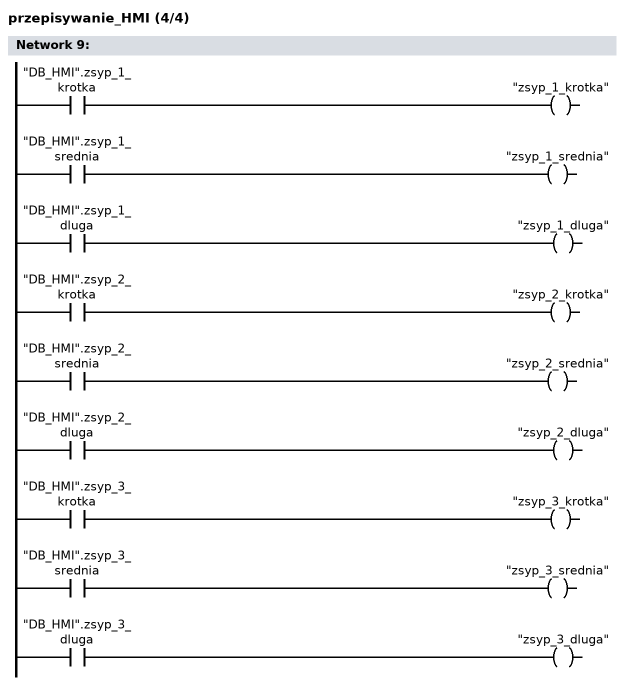
   RUNG wire#powerrail
      Contact( "DB_HMI".zsyp_1_krotka )
      Coil( "zsyp_1_krotka" )
   END_RUNG
   RUNG wire#powerrail
      Contact( "DB_HMI".zsyp_1_srednia )
      Coil( "zsyp_1_srednia" )
   END_RUNG
   RUNG wire#powerrail
      Contact( "DB_HMI".zsyp_1_dluga )
      Coil( "zsyp_1_dluga" )
   END_RUNG
   RUNG wire#powerrail
      Contact( "DB_HMI".zsyp_2_krotka )
      Coil( "zsyp_2_krotka" )
   END_RUNG
   RUNG wire#powerrail
      Contact( "DB_HMI".zsyp_2_srednia )
      Coil( "zsyp_2_srednia" )
   END_RUNG
   RUNG wire#powerrail
      Contact( "DB_HMI".zsyp_2_dluga )
      Coil( "zsyp_2_dluga" )
   END_RUNG
   RUNG wire#powerrail
      Contact( "DB_HMI".zsyp_3_krotka )
      Coil( "zsyp_3_krotka" )
   END_RUNG
   RUNG wire#powerrail
      Contact( "DB_HMI".zsyp_3_srednia )
      Coil( "zsyp_3_srednia" )
   END_RUNG
   RUNG wire#powerrail
      Contact( "DB_HMI".zsyp_3_dluga )
      Coil( "zsyp_3_dluga" )
   END_RUNG
   // the same network as SCL:
   "zsyp_1_krotka" := "DB_HMI".zsyp_1_krotka;
   "zsyp_1_srednia" := "DB_HMI".zsyp_1_srednia;
   "zsyp_1_dluga" := "DB_HMI".zsyp_1_dluga;
   "zsyp_2_krotka" := "DB_HMI".zsyp_2_krotka;
   "zsyp_2_srednia" := "DB_HMI".zsyp_2_srednia;
   "zsyp_2_dluga" := "DB_HMI".zsyp_2_dluga;
   "zsyp_3_krotka" := "DB_HMI".zsyp_3_krotka;
   "zsyp_3_srednia" := "DB_HMI".zsyp_3_srednia;
   "zsyp_3_dluga" := "DB_HMI".zsyp_3_dluga;
END_REGION
END_FUNCTION

FUNCTION "opuszczanie_tartaku" : Void   // FC3, LAD
{ S7_Optimized_Access := 'TRUE' }
VERSION : 0.1
// Wyjazd wagoników z tartaku
BEGIN

REGION Network 1
   // Zapalenie sygnalizatora bocznicy w momencie jej zapełnienia
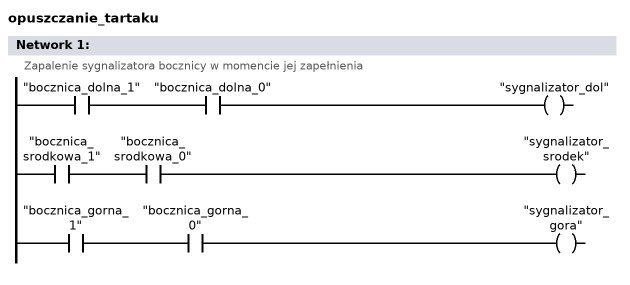
   RUNG wire#powerrail
      Contact( "bocznica_dolna_1" )
      Contact( "bocznica_dolna_0" )
      Coil( "sygnalizator_dol" )
   END_RUNG
   RUNG wire#powerrail
      Contact( "bocznica_srodkowa_1" )
      Contact( "bocznica_srodkowa_0" )
      Coil( "sygnalizator_srodek" )
   END_RUNG
   RUNG wire#powerrail
      Contact( "bocznica_gorna_1" )
      Contact( "bocznica_gorna_0" )
      Coil( "sygnalizator_gora" )
   END_RUNG
   // the same network as SCL:
   "sygnalizator_dol" := "bocznica_dolna_1" AND "bocznica_dolna_0";
   "sygnalizator_srodek" := "bocznica_srodkowa_1" AND "bocznica_srodkowa_0";
   "sygnalizator_gora" := "bocznica_gorna_1" AND "bocznica_gorna_0";
END_REGION
END_FUNCTION

FUNCTION "zmiana_odbiorcy" : Void   // FC4, LAD
{ S7_Optimized_Access := 'TRUE' }
VERSION : 0.1
   VAR_TEMP   // added for the SCL form of the ladder/FBD networks
      _w1 : Bool;
   END_VAR
BEGIN

REGION Network 1: Zmiana trybu normalnego na odbiorcę
   // Przepisywanie wykrytego rozmiaru belki w celu zachowania prawidłowej pracy programu między przełączaniem trybów.
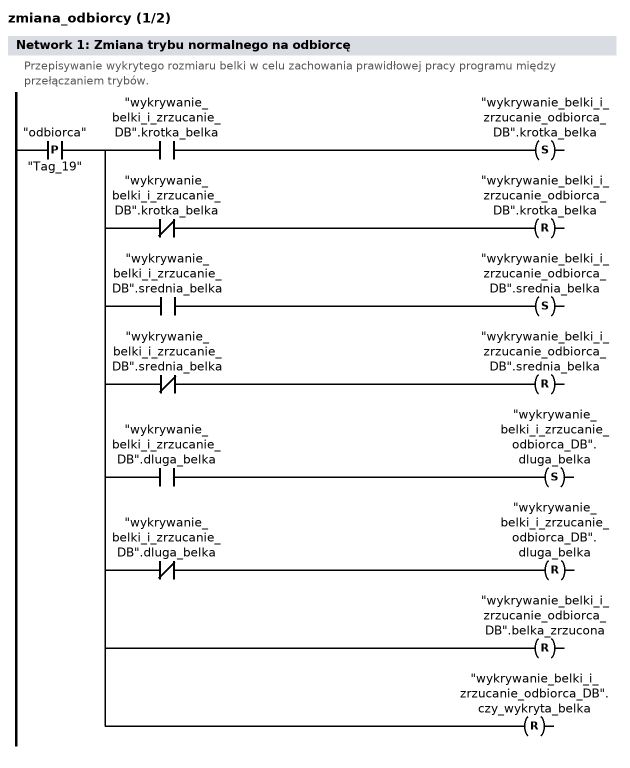
   RUNG wire#powerrail
      P_Contact(operand := "odbiorca", bit := "Tag_19")
      wire#w1
      Contact( "wykrywanie_belki_i_zrzucanie_DB".krotka_belka )
      S_Coil( "wykrywanie_belki_i_zrzucanie_odbiorca_DB".krotka_belka )
   END_RUNG
   RUNG wire#w1
      I_Contact( "wykrywanie_belki_i_zrzucanie_DB".krotka_belka )
      R_Coil( "wykrywanie_belki_i_zrzucanie_odbiorca_DB".krotka_belka )
   END_RUNG
   RUNG wire#w1
      Contact( "wykrywanie_belki_i_zrzucanie_DB".srednia_belka )
      S_Coil( "wykrywanie_belki_i_zrzucanie_odbiorca_DB".srednia_belka )
   END_RUNG
   RUNG wire#w1
      I_Contact( "wykrywanie_belki_i_zrzucanie_DB".srednia_belka )
      R_Coil( "wykrywanie_belki_i_zrzucanie_odbiorca_DB".srednia_belka )
   END_RUNG
   RUNG wire#w1
      Contact( "wykrywanie_belki_i_zrzucanie_DB".dluga_belka )
      S_Coil( "wykrywanie_belki_i_zrzucanie_odbiorca_DB".dluga_belka )
   END_RUNG
   RUNG wire#w1
      I_Contact( "wykrywanie_belki_i_zrzucanie_DB".dluga_belka )
      R_Coil( "wykrywanie_belki_i_zrzucanie_odbiorca_DB".dluga_belka )
   END_RUNG
   RUNG wire#w1
      R_Coil( "wykrywanie_belki_i_zrzucanie_odbiorca_DB".belka_zrzucona )
   END_RUNG
   RUNG wire#w1
      R_Coil( "wykrywanie_belki_i_zrzucanie_odbiorca_DB".czy_wykryta_belka )
   END_RUNG
   // the same network as SCL:
   #_w1 := "odbiorca" AND NOT "Tag_19";   // rising edge of "odbiorca"
   "Tag_19" := "odbiorca";
   IF #_w1 AND "wykrywanie_belki_i_zrzucanie_DB".krotka_belka THEN
       "wykrywanie_belki_i_zrzucanie_odbiorca_DB".krotka_belka := TRUE;
   END_IF;
   IF #_w1 AND NOT "wykrywanie_belki_i_zrzucanie_DB".krotka_belka THEN
       "wykrywanie_belki_i_zrzucanie_odbiorca_DB".krotka_belka := FALSE;
   END_IF;
   IF #_w1 AND "wykrywanie_belki_i_zrzucanie_DB".srednia_belka THEN
       "wykrywanie_belki_i_zrzucanie_odbiorca_DB".srednia_belka := TRUE;
   END_IF;
   IF #_w1 AND NOT "wykrywanie_belki_i_zrzucanie_DB".srednia_belka THEN
       "wykrywanie_belki_i_zrzucanie_odbiorca_DB".srednia_belka := FALSE;
   END_IF;
   IF #_w1 AND "wykrywanie_belki_i_zrzucanie_DB".dluga_belka THEN
       "wykrywanie_belki_i_zrzucanie_odbiorca_DB".dluga_belka := TRUE;
   END_IF;
   IF #_w1 AND NOT "wykrywanie_belki_i_zrzucanie_DB".dluga_belka THEN
       "wykrywanie_belki_i_zrzucanie_odbiorca_DB".dluga_belka := FALSE;
   END_IF;
   IF #_w1 THEN
       "wykrywanie_belki_i_zrzucanie_odbiorca_DB".belka_zrzucona := FALSE;
       "wykrywanie_belki_i_zrzucanie_odbiorca_DB".czy_wykryta_belka := FALSE;
   END_IF;
END_REGION

REGION Network 2: Zmiana z trybu odbiorcy na tryb normalny
   // Przepisywanie wykrytego rozmiaru belki w celu zachowania prawidłowej pracy programu między przełączaniem trybów.
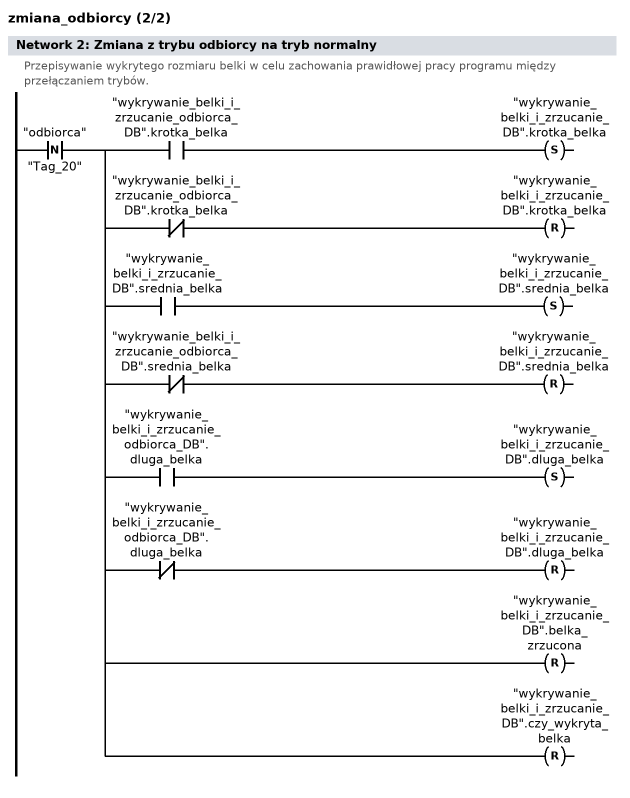
   RUNG wire#powerrail
      N_Contact(operand := "odbiorca", bit := "Tag_20")
      wire#w1
      Contact( "wykrywanie_belki_i_zrzucanie_odbiorca_DB".krotka_belka )
      S_Coil( "wykrywanie_belki_i_zrzucanie_DB".krotka_belka )
   END_RUNG
   RUNG wire#w1
      I_Contact( "wykrywanie_belki_i_zrzucanie_odbiorca_DB".krotka_belka )
      R_Coil( "wykrywanie_belki_i_zrzucanie_DB".krotka_belka )
   END_RUNG
   RUNG wire#w1
      Contact( "wykrywanie_belki_i_zrzucanie_DB".srednia_belka )
      S_Coil( "wykrywanie_belki_i_zrzucanie_DB".srednia_belka )
   END_RUNG
   RUNG wire#w1
      I_Contact( "wykrywanie_belki_i_zrzucanie_odbiorca_DB".srednia_belka )
      R_Coil( "wykrywanie_belki_i_zrzucanie_DB".srednia_belka )
   END_RUNG
   RUNG wire#w1
      Contact( "wykrywanie_belki_i_zrzucanie_odbiorca_DB".dluga_belka )
      S_Coil( "wykrywanie_belki_i_zrzucanie_DB".dluga_belka )
   END_RUNG
   RUNG wire#w1
      I_Contact( "wykrywanie_belki_i_zrzucanie_odbiorca_DB".dluga_belka )
      R_Coil( "wykrywanie_belki_i_zrzucanie_DB".dluga_belka )
   END_RUNG
   RUNG wire#w1
      R_Coil( "wykrywanie_belki_i_zrzucanie_DB".belka_zrzucona )
   END_RUNG
   RUNG wire#w1
      R_Coil( "wykrywanie_belki_i_zrzucanie_DB".czy_wykryta_belka )
   END_RUNG
   // the same network as SCL:
   #_w1 := NOT "odbiorca" AND "Tag_20";   // falling edge of "odbiorca"
   "Tag_20" := "odbiorca";
   IF #_w1 AND "wykrywanie_belki_i_zrzucanie_odbiorca_DB".krotka_belka THEN
       "wykrywanie_belki_i_zrzucanie_DB".krotka_belka := TRUE;
   END_IF;
   IF #_w1 AND NOT "wykrywanie_belki_i_zrzucanie_odbiorca_DB".krotka_belka THEN
       "wykrywanie_belki_i_zrzucanie_DB".krotka_belka := FALSE;
   END_IF;
   IF #_w1 AND "wykrywanie_belki_i_zrzucanie_DB".srednia_belka THEN
       "wykrywanie_belki_i_zrzucanie_DB".srednia_belka := TRUE;
   END_IF;
   IF #_w1 AND NOT "wykrywanie_belki_i_zrzucanie_odbiorca_DB".srednia_belka THEN
       "wykrywanie_belki_i_zrzucanie_DB".srednia_belka := FALSE;
   END_IF;
   IF #_w1 AND "wykrywanie_belki_i_zrzucanie_odbiorca_DB".dluga_belka THEN
       "wykrywanie_belki_i_zrzucanie_DB".dluga_belka := TRUE;
   END_IF;
   IF #_w1 AND NOT "wykrywanie_belki_i_zrzucanie_odbiorca_DB".dluga_belka THEN
       "wykrywanie_belki_i_zrzucanie_DB".dluga_belka := FALSE;
   END_IF;
   IF #_w1 THEN
       "wykrywanie_belki_i_zrzucanie_DB".belka_zrzucona := FALSE;
       "wykrywanie_belki_i_zrzucanie_DB".czy_wykryta_belka := FALSE;
   END_IF;
END_REGION
END_FUNCTION

ORGANIZATION_BLOCK "Main"   // OB1, LAD, ProgramCycle
TITLE = "Main Program Sweep (Cycle)"
{ S7_Optimized_Access := 'TRUE' }
VERSION : 0.1
// Główny program projektu wywołujący poszczególne bloki FC i FB.
   VAR_INPUT
      Initial_Call : Bool;   // Initial call of this OB
      Remanence : Bool;   // =True, if remanent data are available
   END_VAR
BEGIN

REGION Network 1
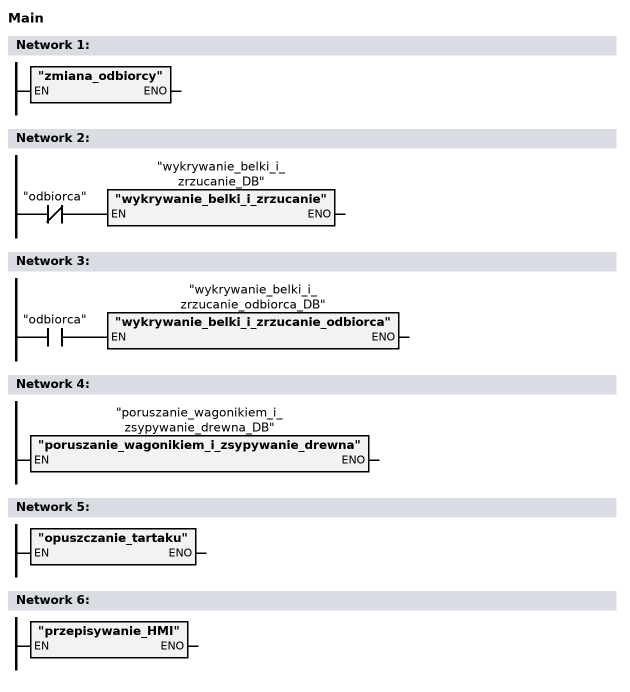
   RUNG wire#powerrail
      "zmiana_odbiorcy"()
   END_RUNG
   // the same network as SCL:
   "zmiana_odbiorcy"();
END_REGION

REGION Network 2
   RUNG wire#powerrail
      I_Contact( "odbiorca" )
      "wykrywanie_belki_i_zrzucanie_DB"()
   END_RUNG
   // the same network as SCL:
   IF NOT "odbiorca" THEN
       "wykrywanie_belki_i_zrzucanie_DB"();   // "wykrywanie_belki_i_zrzucanie"
   END_IF;
END_REGION

REGION Network 3
   RUNG wire#powerrail
      Contact( "odbiorca" )
      "wykrywanie_belki_i_zrzucanie_odbiorca_DB"()
   END_RUNG
   // the same network as SCL:
   IF "odbiorca" THEN
       "wykrywanie_belki_i_zrzucanie_odbiorca_DB"();   // "wykrywanie_belki_i_zrzucanie_odbiorca"
   END_IF;
END_REGION

REGION Network 4
   RUNG wire#powerrail
      "poruszanie_wagonikiem_i_zsypywanie_drewna_DB"()
   END_RUNG
   // the same network as SCL:
   "poruszanie_wagonikiem_i_zsypywanie_drewna_DB"();   // "poruszanie_wagonikiem_i_zsypywanie_drewna"
END_REGION

REGION Network 5
   RUNG wire#powerrail
      "opuszczanie_tartaku"()
   END_RUNG
   // the same network as SCL:
   "opuszczanie_tartaku"();
END_REGION

REGION Network 6
   RUNG wire#powerrail
      "przepisywanie_HMI"()
   END_RUNG
   // the same network as SCL:
   "przepisywanie_HMI"();
END_REGION
END_ORGANIZATION_BLOCK

(* ===== HMI "HMI_RT_2" =====
system functions are stored by id; their names below are inferred from use
connection "HMI_Connection_1": ETHERNET, S7_1200_OMS

HMI tags "Default tag table"
   "Tag_ScreenNumber" : UInt, internal
   "DB_HMI_napelnienie_zsyp_krotki" : Bool = PLC DB_HMI.napelnienie_zsyp_krotki, 100 ms
   "DB_HMI_napelnienie_zsyp_sredni" : Bool = PLC DB_HMI.napelnienie_zsyp_sredni, 100 ms
   "DB_HMI_napelnienie_zsyp_dlugi" : Bool = PLC DB_HMI.napelnienie_zsyp_dlugi, 100 ms
   "DB_HMI_oproznianie_zsyp_krotki" : Bool = PLC DB_HMI.oproznianie_zsyp_krotki, 100 ms
   "DB_HMI_oproznianie_zsyp_sredni" : Bool = PLC DB_HMI.oproznianie_zsyp_sredni, 100 ms
   "DB_HMI_oproznianie_zsyp_dlugi" : Bool = PLC DB_HMI.oproznianie_zsyp_dlugi, 100 ms
   "DB_HMI_status_ruchu_wagonika" : Bool = PLC DB_HMI.status_ruchu_wagonika, 100 ms
   "DB_HMI_wagonik_dlugi" : Bool = PLC DB_HMI.wagonik_dlugi, 100 ms
   "DB_HMI_wagonik_sredni" : Bool = PLC DB_HMI.wagonik_sredni, 100 ms
   "DB_HMI_wagonik_krotki" : Bool = PLC DB_HMI.wagonik_krotki, 100 ms
   "DB_HMI_zapelnienie_bocznicy_dlugiej" : Byte = PLC DB_HMI.zapelnienie_bocznicy_dlugiej, 100 ms
   "DB_HMI_sygnalizator_bocznica_srednia" : Bool = PLC DB_HMI.sygnalizator_bocznica_srednia, 100 ms
   "DB_HMI_zapelnienie_bocznicy_sredniej" : Byte = PLC DB_HMI.zapelnienie_bocznicy_sredniej, 100 ms
   "DB_HMI_zapelnienie_bocznicy_krotkiej" : Byte = PLC DB_HMI.zapelnienie_bocznicy_krotkiej, 100 ms
   "DB_HMI_sygnalizator_bocznica_dluga" : Bool = PLC DB_HMI.sygnalizator_bocznica_dluga, 100 ms
   "DB_HMI_sygnalizator_bocznica_krotka" : Bool = PLC DB_HMI.sygnalizator_bocznica_krotka, 100 ms
   "DB_HMI_ustawienie_zwrotnicy" : Byte = PLC DB_HMI.ustawienie_zwrotnicy, 100 ms
   "DB_HMI_odbiorca" : Bool = PLC DB_HMI.odbiorca AT %DB1.DBW0, 100 ms
   "DB_HMI_belka_krotka" : Bool = PLC DB_HMI.belka_krotka AT %DB1.DBX0.0, 100 ms
   "DB_HMI_belka_srednia" : Bool = PLC DB_HMI.belka_srednia AT %DB1.DBX0.0, 100 ms
   "DB_HMI_belka_dluga" : Bool = PLC DB_HMI.belka_dluga AT %DB1.DBX0.0, 100 ms
   "DB_HMI_zsyp_1_krotka" : Bool = PLC DB_HMI.zsyp_1_krotka, 100 ms
   "DB_HMI_zsyp_1_srednia" : Bool = PLC DB_HMI.zsyp_1_srednia, 100 ms
   "DB_HMI_zsyp_1_dluga" : Bool = PLC DB_HMI.zsyp_1_dluga, 100 ms
   "DB_HMI_zsyp_2_krotka" : Bool = PLC DB_HMI.zsyp_2_krotka, 100 ms
   "DB_HMI_zsyp_2_srednia" : Bool = PLC DB_HMI.zsyp_2_srednia, 100 ms
   "DB_HMI_zsyp_2_dluga" : Bool = PLC DB_HMI.zsyp_2_dluga, 100 ms
   "DB_HMI_zsyp_3_krotka" : Bool = PLC DB_HMI.zsyp_3_krotka, 100 ms
   "DB_HMI_zsyp_3_srednia" : Bool = PLC DB_HMI.zsyp_3_srednia, 100 ms
   "DB_HMI_zsyp_3_dluga" : Bool = PLC DB_HMI.zsyp_3_dluga, 100 ms

screen "Root screen" 800x420, template "Template_1"
   on GenerateScreen: SetTag("Tag_ScreenNumber", 1)
   GraphicIOField "PlotLight_Square_G" at 668,266 size 30x30; PictureOff "PilotLight_Square_G_Off_256c"; PictureOn "PilotLight_Square_G_On_256c"
      ProcessValue <- "DB_HMI_status_ruchu_wagonika"
   TextField "Text field_4" at 10,9 size 224x23; Text 'Rozmiar wykrytej belki:'
   Switch "Lever_Vertical_2" at 726,48 size 38x62; CaptionText 'Switch'; TextOff '0'; TextOn '1'; PictureOff "Lever_Vertical_2_Off_256c"; PictureOn "Lever_Vertical_2_On_256c"
      on Change: "Aktualizacja_nazw"()
      ProcessValue <- "DB_HMI_odbiorca"
   TextField "Text field_5" at 682,5 size 117x42; Text 'Uniwersalny Odbiorca'
   Switch "l_dl" at 413,77 size 30x30; CaptionText 'Switch'; TextOff '0'; TextOn '1'; PictureOff "Pushbutton_Round_G_Off_256c"; PictureOn "Pushbutton_Round_G_On_256c"
      Visibility <- "DB_HMI_odbiorca"
      on SwitchOn: "Przypisanie_belki_do_zsypu"('dluga', 'lewy')
      on SwitchOff: "Odpiecie_belki_do_zsypu"('dluga', 'lewy')
      ProcessValue <- "DB_HMI_zsyp_1_dluga"
   Switch "l_sr" at 413,45 size 30x30; CaptionText 'Switch'; TextOff '0'; TextOn '1'; PictureOff "Pushbutton_Round_R_Off_256c"; PictureOn "Pushbutton_Round_R_On_256c"
      Visibility <- "DB_HMI_odbiorca"
      on SwitchOn: "Przypisanie_belki_do_zsypu"('srednia', 'lewy')
      on SwitchOff: "Odpiecie_belki_do_zsypu"('srednia', 'lewy')
      ProcessValue <- "DB_HMI_zsyp_1_srednia"
   Switch "l_kr" at 413,12 size 30x30; CaptionText 'Switch'; TextOff '0'; TextOn '1'; PictureOff "Pushbutton_Round_RN_Off_256c"; PictureOn "Pushbutton_Round_RN_On_256c"
      Visibility <- "DB_HMI_odbiorca"
      on SwitchOn: "Przypisanie_belki_do_zsypu"('krotka', 'lewy')
      on SwitchOff: "Odpiecie_belki_do_zsypu"('krotka', 'lewy')
      ProcessValue <- "DB_HMI_zsyp_1_krotka"
   Switch "s_dl" at 516,79 size 30x30; CaptionText 'Switch'; TextOff '0'; TextOn '1'; PictureOff "Pushbutton_Round_G_Off_256c"; PictureOn "Pushbutton_Round_G_On_256c"
      Visibility <- "DB_HMI_odbiorca"
      ProcessValue <- "DB_HMI_zsyp_2_dluga"
      on SwitchOn: "Przypisanie_belki_do_zsypu"('dluga', 'srodkowy')
      on SwitchOff: "Odpiecie_belki_do_zsypu"('dluga', 'srodkowy')
   Switch "s_sr" at 516,47 size 30x30; CaptionText 'Switch'; TextOff '0'; TextOn '1'; PictureOff "Pushbutton_Round_R_Off_256c"; PictureOn "Pushbutton_Round_R_On_256c"
      Visibility <- "DB_HMI_odbiorca"
      ProcessValue <- "DB_HMI_zsyp_2_srednia"
      on SwitchOn: "Przypisanie_belki_do_zsypu"('srednia', 'srodkowy')
      on SwitchOff: "Odpiecie_belki_do_zsypu"('srednia', 'srodkowy')
   Switch "s_kr" at 516,14 size 30x30; CaptionText 'Switch'; TextOff '0'; TextOn '1'; PictureOff "Pushbutton_Round_RN_Off_256c"; PictureOn "Pushbutton_Round_RN_On_256c"
      Visibility <- "DB_HMI_odbiorca"
      on SwitchOn: "Przypisanie_belki_do_zsypu"('krotka', 'srodkowy')
      on SwitchOff: "Odpiecie_belki_do_zsypu"('krotka', 'srodkowy')
      ProcessValue <- "DB_HMI_zsyp_2_krotka"
   Switch "p_dl" at 617,81 size 30x30; CaptionText 'Switch'; TextOff '0'; TextOn '1'; PictureOff "Pushbutton_Round_G_Off_256c"; PictureOn "Pushbutton_Round_G_On_256c"
      Visibility <- "DB_HMI_odbiorca"
      ProcessValue <- "DB_HMI_zsyp_3_dluga"
      on SwitchOn: "Przypisanie_belki_do_zsypu"('dluga', 'prawy')
      on SwitchOff: "Odpiecie_belki_do_zsypu"('dluga', 'prawy')
   Switch "p_sr" at 617,49 size 30x30; CaptionText 'Switch'; TextOff '0'; TextOn '1'; PictureOff "Pushbutton_Round_R_Off_256c"; PictureOn "Pushbutton_Round_R_On_256c"
      Visibility <- "DB_HMI_odbiorca"
      ProcessValue <- "DB_HMI_zsyp_3_srednia"
      on SwitchOn: "Przypisanie_belki_do_zsypu"('srednia', 'prawy')
      on SwitchOff: "Odpiecie_belki_do_zsypu"('srednia', 'prawy')
   Switch "p_kr" at 617,16 size 30x30; CaptionText 'Switch'; TextOff '0'; TextOn '1'; PictureOff "Pushbutton_Round_RN_Off_256c"; PictureOn "Pushbutton_Round_RN_On_256c"
      Visibility <- "DB_HMI_odbiorca"
      ProcessValue <- "DB_HMI_zsyp_3_krotka"
      on SwitchOn: "Przypisanie_belki_do_zsypu"('krotka', 'prawy')
      on SwitchOff: "Odpiecie_belki_do_zsypu"('krotka', 'prawy')
   GraphicIOField "PlotLight_Round_G_6" at 10,34 size 25x25; PictureOn "PilotLight_Round_G_On_256c"; PictureOff "PilotLight_Round_G_Off_256c"
      ProcessValue <- "DB_HMI_belka_krotka"
   GraphicIOField "PlotLight_Round_G_7" at 10,64 size 25x25; PictureOff "PilotLight_Round_G_Off_256c"; PictureOn "PilotLight_Round_G_On_256c"
      ProcessValue <- "DB_HMI_belka_srednia"
   GraphicIOField "PlotLight_Round_G_8" at 10,94 size 25x25; PictureOn "PilotLight_Round_G_On_256c"; PictureOff "PilotLight_Round_G_Off_256c"
      ProcessValue <- "DB_HMI_belka_dluga"
   TextField "Text field_6" at 43,37 size 60x23; Text 'krótki'
   TextField "Text field_7" at 43,65 size 61x23; Text 'średni'
   TextField "Text field_8" at 45,95 size 50x23; Text 'długi'
   SymbolLibrary "Symbol library_3" at 600,114 size 67x91
      Appearance <- "DB_HMI_napelnienie_zsyp_dlugi"
   SymbolLibrary "Symbol library_2" at 498,114 size 67x91
      Appearance <- "DB_HMI_napelnienie_zsyp_sredni"
   SymbolLibrary "Symbol library_1" at 396,114 size 67x91
      Appearance <- "DB_HMI_napelnienie_zsyp_krotki"
   GraphicIOField "PlotLight_Round_G" at 419,180 size 20x19; PictureOff "PilotLight_Round_G_Off_256c"; PictureOn "PilotLight_Round_G_On_256c"
      ProcessValue <- "DB_HMI_oproznianie_zsyp_krotki"
   GraphicIOField "PlotLight_Round_G_1" at 521,180 size 20x19; PictureOn "PilotLight_Round_G_On_256c"; PictureOff "PilotLight_Round_G_Off_256c"
      ProcessValue <- "DB_HMI_oproznianie_zsyp_sredni"
   GraphicIOField "PlotLight_Round_G_2" at 623,179 size 20x19; PictureOff "PilotLight_Round_G_Off_256c"; PictureOn "PilotLight_Round_G_On_256c"
      ProcessValue <- "DB_HMI_napelnienie_zsyp_dlugi"
   GraphicView "Graphic view_4" at 594,210 size 74x65; Picture "Graphic_5"
      Visibility <- "DB_HMI_wagonik_dlugi"
   GraphicView "Graphic view_5" at 494,210 size 74x65; Picture "Graphic_5"
      Visibility <- "DB_HMI_wagonik_sredni"
   GraphicView "Graphic view_6" at 392,210 size 74x65; Picture "Graphic_5"
      Visibility <- "DB_HMI_wagonik_krotki"
   GraphicView "Graphic view_7" at 90,156 size 58x55; Picture "Graphic_5"
      Visibility <- "DB_HMI_zapelnienie_bocznicy_dlugiej"
   GraphicView "Graphic view_8" at 160,156 size 58x55; Picture "Graphic_5"
      Visibility <- "DB_HMI_zapelnienie_bocznicy_dlugiej"
   GraphicView "Graphic view_9" at 91,222 size 58x55; Picture "Graphic_5"
      Visibility <- "DB_HMI_zapelnienie_bocznicy_sredniej"
   GraphicView "Graphic view_10" at 161,222 size 58x55; Picture "Graphic_5"
      Visibility <- "DB_HMI_zapelnienie_bocznicy_sredniej"
   GraphicView "Graphic view_11" at 90,291 size 58x55; Picture "Graphic_5"
      Visibility <- "DB_HMI_zapelnienie_bocznicy_krotkiej"
   GraphicView "Graphic view_12" at 160,291 size 58x55; Picture "Graphic_5"
      Visibility <- "DB_HMI_zapelnienie_bocznicy_krotkiej"
   Line "Line_5" at 229,212 size 77x67
      Visibility <- "DB_HMI_ustawienie_zwrotnicy"
   Line "Line_6" at 230,279 size 75x0
      Visibility <- "DB_HMI_ustawienie_zwrotnicy"
   Line "Line_7" at 228,280 size 77x68
      Visibility <- "DB_HMI_ustawienie_zwrotnicy"
   GraphicIOField "PlotLight_Round_G_3" at 59,156 size 26x24; PictureOff "PilotLight_Round_G_Off_256c"; PictureOn "PilotLight_Round_G_On_256c"
      ProcessValue <- "DB_HMI_sygnalizator_bocznica_dluga"
   GraphicIOField "PlotLight_Round_G_4" at 57,221 size 26x24; PictureOn "PilotLight_Round_G_On_256c"; PictureOff "PilotLight_Round_G_Off_256c"
      ProcessValue <- "DB_HMI_sygnalizator_bocznica_srednia"
   GraphicIOField "PlotLight_Round_G_5" at 57,290 size 26x24; PictureOff "PilotLight_Round_G_Off_256c"; PictureOn "PilotLight_Round_G_On_256c"
      ProcessValue <- "DB_HMI_sygnalizator_bocznica_krotka"
   TextField "tekst_zsyp_lewy" at 393,117 size 72x54; Text 'pnie -----'
   TextField "tekst_zsyp_srodkowy" at 496,120 size 69x50; Text 'pnie -----'
   TextField "tekst_zsyp_prawy" at 600,118 size 68x54; Text 'pnie -----'
   TextField "Text field_9" at 330,48 size 74x23; Text 'Średnie'
      Visibility <- "DB_HMI_odbiorca"
   TextField "Text field_10" at 331,79 size 63x23; Text 'Długie'
      Visibility <- "DB_HMI_odbiorca"
   TextField "Text field_11" at 331,17 size 72x23; Text 'Krótkie'
      Visibility <- "DB_HMI_odbiorca"

Template "Template_1" 800x420
   Button "Exit" at 720,360 size 78x58; TextOn 'Exit'; TextOff 'Exit'; PictureOn "ExitRuntime_TP700_Comfort_TR"; PictureOff "ExitRuntime_TP700_Comfort_TR"
      on Release: StopRuntime(0)
   Button "Template_Button" at 640,360 size 78x58; TextOff 'Text'
   Button "Template_Button_1" at 560,360 size 78x58; TextOff 'Text'
   Button "Template_Button_2" at 480,360 size 78x58; TextOff 'Text'
   Button "Template_Button_3" at 400,360 size 78x58; TextOff 'Text'
   Button "Template_Button_4" at 321,360 size 78x58; TextOff 'Text'
   Button "Template_Button_5" at 241,360 size 78x58; TextOff 'Text'
   Button "Template_Button_6" at 161,360 size 78x58; TextOff 'Text'
   Button "Template_Button_7" at 81,360 size 78x58; TextOff 'Text'
   Button "Start screen" at 1,360 size 78x58; TextOn 'Start screen'; TextOff 'Start screen'; PictureOn "NavigateHome_TP700_Comfort_TR"; PictureOff "NavigateHome_TP700_Comfort_TR"
      on Release: ActivateScreen("Root screen", 0)

VB script "Przypisanie_belki_do_zsypu"
   'Skrypt ustawiający odpowiednie napisy na zsypach w zależności od wybranego przycisku oraz blokowanie pozostałych wyborów.
   'Zsyp: 				1		2		3
   'Rozmiar belki:		1_kr	s_kr	p_kr
   '					1_sr	s_sr	p_sr
   '					1_dl	s_dl	p_dl
   
   If zsyp = "lewy" Then
   	If dlugosc_belki = "krotka" Then	'jezeli wybrano rozmiar belki krotki
   		HmiRuntime.Screens("Root screen").ScreenItems("tekst_zsyp_lewy").Text = "pnie" & Chr(10) & "krótkie"	'ustaw na zsypie informacje o wybranej belce 
   		HmiRuntime.Screens("Root screen").ScreenItems("l_sr").Enabled = False
   		HmiRuntime.Screens("Root screen").ScreenItems("l_dl").Enabled = False							
   		HmiRuntime.Screens("Root screen").ScreenItems("s_kr").Enabled = False							
   		HmiRuntime.Screens("Root screen").ScreenItems("p_kr").Enabled = False
   	ElseIf dlugosc_belki = "srednia" Then
   		HmiRuntime.Screens("Root screen").ScreenItems("tekst_zsyp_lewy").Text = "pnie" & Chr(10) & "średnie" 
   		HmiRuntime.Screens("Root screen").ScreenItems("l_kr").Enabled = False
   		HmiRuntime.Screens("Root screen").ScreenItems("l_dl").Enabled = False
   		HmiRuntime.Screens("Root screen").ScreenItems("s_sr").Enabled = False
   		HmiRuntime.Screens("Root screen").ScreenItems("p_sr").Enabled = False
   	ElseIf dlugosc_belki = "dluga" Then
   		HmiRuntime.Screens("Root screen").ScreenItems("tekst_zsyp_lewy").Text = "pnie" & Chr(10) & "długie" 
   		HmiRuntime.Screens("Root screen").ScreenItems("l_kr").Enabled = False
   		HmiRuntime.Screens("Root screen").ScreenItems("l_sr").Enabled = False
   		HmiRuntime.Screens("Root screen").ScreenItems("s_dl").Enabled = False
   		HmiRuntime.Screens("Root screen").ScreenItems("p_dl").Enabled = False
   	End If
   ElseIf zsyp = "srodkowy" Then
   	If dlugosc_belki = "krotka" Then
   		HmiRuntime.Screens("Root screen").ScreenItems("tekst_zsyp_srodkowy").Text = "pnie" & Chr(10) & "krótkie" 
   		HmiRuntime.Screens("Root screen").ScreenItems("s_sr").Enabled = False
   		HmiRuntime.Screens("Root screen").ScreenItems("s_dl").Enabled = False
   		HmiRuntime.Screens("Root screen").ScreenItems("l_kr").Enabled = False
   		HmiRuntime.Screens("Root screen").ScreenItems("p_kr").Enabled = False
   	ElseIf dlugosc_belki = "srednia" Then
   		HmiRuntime.Screens("Root screen").ScreenItems("tekst_zsyp_srodkowy").Text = "pnie" & Chr(10) & "średnie" 
   		HmiRuntime.Screens("Root screen").ScreenItems("s_kr").Enabled = False
   		HmiRuntime.Screens("Root screen").ScreenItems("s_dl").Enabled = False
   		HmiRuntime.Screens("Root screen").ScreenItems("l_sr").Enabled = False
   		HmiRuntime.Screens("Root screen").ScreenItems("p_sr").Enabled = False
   	ElseIf dlugosc_belki = "dluga" Then
   		HmiRuntime.Screens("Root screen").ScreenItems("tekst_zsyp_srodkowy").Text = "pnie" & Chr(10) & "długie" 
   		HmiRuntime.Screens("Root screen").ScreenItems("s_kr").Enabled = False
   		HmiRuntime.Screens("Root screen").ScreenItems("s_sr").Enabled = False
   		HmiRuntime.Screens("Root screen").ScreenItems("l_dl").Enabled = False
   		HmiRuntime.Screens("Root screen").ScreenItems("p_dl").Enabled = False
   	End If
   ElseIf zsyp = "prawy" Then
   	If dlugosc_belki = "krotka" Then
   		HmiRuntime.Screens("Root screen").ScreenItems("tekst_zsyp_prawy").Text = "pnie" & Chr(10) & "krótkie" 
   		HmiRuntime.Screens("Root screen").ScreenItems("p_sr").Enabled = False
   		HmiRuntime.Screens("Root screen").ScreenItems("p_dl").Enabled = False
   		HmiRuntime.Screens("Root screen").ScreenItems("l_kr").Enabled = False
   		HmiRuntime.Screens("Root screen").ScreenItems("s_kr").Enabled = False
   	ElseIf dlugosc_belki = "srednia" Then
   		HmiRuntime.Screens("Root screen").ScreenItems("tekst_zsyp_prawy").Text = "pnie" & Chr(10) & "średnie" 
   		HmiRuntime.Screens("Root screen").ScreenItems("p_kr").Enabled = False
   		HmiRuntime.Screens("Root screen").ScreenItems("p_dl").Enabled = False
   		HmiRuntime.Screens("Root screen").ScreenItems("l_sr").Enabled = False
   		HmiRuntime.Screens("Root screen").ScreenItems("s_sr").Enabled = False
   	ElseIf dlugosc_belki = "dluga" Then
   		HmiRuntime.Screens("Root screen").ScreenItems("tekst_zsyp_prawy").Text = "pnie" & Chr(10) & "długie" 
   		HmiRuntime.Screens("Root screen").ScreenItems("p_kr").Enabled = False
   		HmiRuntime.Screens("Root screen").ScreenItems("p_sr").Enabled = False
   		HmiRuntime.Screens("Root screen").ScreenItems("l_dl").Enabled = False
   		HmiRuntime.Screens("Root screen").ScreenItems("s_dl").Enabled = False
   	End If
   End If

VB script "Odpiecie_belki_do_zsypu"
   'Skrypt realizujący odblokowywanie pozostałych przycisków w momencie odklikania danego przycisku
   
   If zsyp = "lewy" Then
   	If dlugosc_belki = "krotka" Then
   		HmiRuntime.Screens("Root screen").ScreenItems("tekst_zsyp_lewy").Text = "pnie" & Chr(10) & "-----" 
   		If Not SmartTags("DB_HMI_zsyp_3_srednia") And Not SmartTags("DB_HMI_zsyp_2_srednia") Then
   			HmiRuntime.Screens("Root screen").ScreenItems("l_sr").Enabled = True							
   		End If
   		If Not SmartTags("DB_HMI_zsyp_3_dluga") And Not SmartTags("DB_HMI_zsyp_2_dluga") Then
   			HmiRuntime.Screens("Root screen").ScreenItems("l_dl").Enabled = True
   		End If
   		If Not SmartTags("DB_HMI_zsyp_2_srednia") And Not SmartTags("DB_HMI_zsyp_2_dluga") Then							
   			HmiRuntime.Screens("Root screen").ScreenItems("s_kr").Enabled = True
   		End If
   		If Not SmartTags("DB_HMI_zsyp_3_srednia") And Not SmartTags("DB_HMI_zsyp_3_dluga") Then
   			HmiRuntime.Screens("Root screen").ScreenItems("p_kr").Enabled = True
   		End If							
   	ElseIf dlugosc_belki = "srednia" Then
   		HmiRuntime.Screens("Root screen").ScreenItems("tekst_zsyp_lewy").Text = "pnie" & Chr(10) & "-----"
   		If Not SmartTags("DB_HMI_zsyp_2_krotka") And Not SmartTags("DB_HMI_zsyp_3_krotka") Then
   			HmiRuntime.Screens("Root screen").ScreenItems("l_kr").Enabled = True
   		End If
   		If Not SmartTags("DB_HMI_zsyp_2_dluga") And Not SmartTags("DB_HMI_zsyp_3_dluga") Then
   			HmiRuntime.Screens("Root screen").ScreenItems("l_dl").Enabled = True
   		End If
   		If Not SmartTags("DB_HMI_zsyp_2_krotka") And Not SmartTags("DB_HMI_zsyp_2_dluga") Then
   			HmiRuntime.Screens("Root screen").ScreenItems("s_sr").Enabled = True
   		End If
   		If Not SmartTags("DB_HMI_zsyp_3_krotka") And Not SmartTags("DB_HMI_zsyp_3_dluga") Then
   			HmiRuntime.Screens("Root screen").ScreenItems("p_sr").Enabled = True
   		End If
   	ElseIf dlugosc_belki = "dluga" Then
   		HmiRuntime.Screens("Root screen").ScreenItems("tekst_zsyp_lewy").Text = "pnie" & Chr(10) & "-----" 
   		If Not SmartTags("DB_HMI_zsyp_2_krotka") And Not SmartTags("DB_HMI_zsyp_3_krotka") Then
   			HmiRuntime.Screens("Root screen").ScreenItems("l_kr").Enabled = True
   		End If
   		If Not SmartTags("DB_HMI_zsyp_2_srednia") And Not SmartTags("DB_HMI_zsyp_3_srednia") Then
   			HmiRuntime.Screens("Root screen").ScreenItems("l_sr").Enabled = True
   		End If
   		If Not SmartTags("DB_HMI_zsyp_2_krotka") And Not SmartTags("DB_HMI_zsyp_2_srednia") Then
   			HmiRuntime.Screens("Root screen").ScreenItems("s_dl").Enabled = True
   		End If
   		If Not SmartTags("DB_HMI_zsyp_3_krotka") And Not SmartTags("DB_HMI_zsyp_3_srednia") Then
   			HmiRuntime.Screens("Root screen").ScreenItems("p_dl").Enabled = True
   		End If
   	End If
   ElseIf zsyp = "srodkowy" Then
   	If dlugosc_belki = "krotka" Then
   		HmiRuntime.Screens("Root screen").ScreenItems("tekst_zsyp_srodkowy").Text = "pnie" & Chr(10) & "-----"
   		If Not SmartTags("DB_HMI_zsyp_2_srednia") And Not SmartTags("DB_HMI_zsyp_3_srednia") Then
   			HmiRuntime.Screens("Root screen").ScreenItems("s_sr").Enabled = True
   		End If
   		If Not SmartTags("DB_HMI_zsyp_1_dluga") And Not SmartTags("DB_HMI_zsyp_3_dluga") Then
   			HmiRuntime.Screens("Root screen").ScreenItems("s_dl").Enabled = True
   		End If
   		If Not SmartTags("DB_HMI_zsyp_1_srednia") And Not SmartTags("DB_HMI_zsyp_1_dluga") Then
   			HmiRuntime.Screens("Root screen").ScreenItems("l_kr").Enabled = True
   		End If
   		If Not SmartTags("DB_HMI_zsyp_3_srednia") And Not SmartTags("DB_HMI_zsyp_3_dluga") Then
   			HmiRuntime.Screens("Root screen").ScreenItems("p_kr").Enabled = True
   		End If
   	ElseIf dlugosc_belki = "srednia" Then
   		HmiRuntime.Screens("Root screen").ScreenItems("tekst_zsyp_srodkowy").Text = "pnie" & Chr(10) & "-----" 
   		If Not SmartTags("DB_HMI_zsyp_1_krotka") And Not SmartTags("DB_HMI_zsyp_3_krotka") Then
   			HmiRuntime.Screens("Root screen").ScreenItems("s_kr").Enabled = True
   		End If
   		If Not SmartTags("DB_HMI_zsyp_1_dluga") And Not SmartTags("DB_HMI_zsyp_3_dluga") Then
   			HmiRuntime.Screens("Root screen").ScreenItems("s_dl").Enabled = True
   		End If
   		If Not SmartTags("DB_HMI_zsyp_1_krotka") And Not SmartTags("DB_HMI_zsyp_1_dluga") Then
   			HmiRuntime.Screens("Root screen").ScreenItems("l_sr").Enabled = True
   		End If
   		If Not SmartTags("DB_HMI_zsyp_3_krotka") And Not SmartTags("DB_HMI_zsyp_3_dluga") Then
   			HmiRuntime.Screens("Root screen").ScreenItems("p_sr").Enabled = True
   		End If
   	ElseIf dlugosc_belki = "dluga" Then
   		HmiRuntime.Screens("Root screen").ScreenItems("tekst_zsyp_srodkowy").Text = "pnie" & Chr(10) & "-----"
   		If Not SmartTags("DB_HMI_zsyp_1_krotka") And Not SmartTags("DB_HMI_zsyp_3_krotka") Then
   			HmiRuntime.Screens("Root screen").ScreenItems("s_kr").Enabled = True
   		End If
   		If Not SmartTags("DB_HMI_zsyp_1_srednia") And Not SmartTags("DB_HMI_zsyp_3_srednia") Then
   			HmiRuntime.Screens("Root screen").ScreenItems("s_sr").Enabled = True
   		End If
   		If Not SmartTags("DB_HMI_zsyp_1_krotka") And Not SmartTags("DB_HMI_zsyp_1_srednia") Then
   			HmiRuntime.Screens("Root screen").ScreenItems("l_dl").Enabled = True
   		End If
   		If Not SmartTags("DB_HMI_zsyp_3_krotka") And Not SmartTags("DB_HMI_zsyp_3_srednia") Then
   			HmiRuntime.Screens("Root screen").ScreenItems("p_dl").Enabled = True
   		End If
   	End If
   ElseIf zsyp = "prawy" Then
   	If dlugosc_belki = "krotka" Then
   		HmiRuntime.Screens("Root screen").ScreenItems("tekst_zsyp_prawy").Text = "pnie" & Chr(10) & "-----"
   		If Not SmartTags("DB_HMI_zsyp_1_srednia") And Not SmartTags("DB_HMI_zsyp_2_srednia") Then
   			HmiRuntime.Screens("Root screen").ScreenItems("p_sr").Enabled = True
   		End If
   		If Not SmartTags("DB_HMI_zsyp_1_dluga") And Not SmartTags("DB_HMI_zsyp_2_dluga") Then
   			HmiRuntime.Screens("Root screen").ScreenItems("p_dl").Enabled = True
   		End If
   		If Not SmartTags("DB_HMI_zsyp_1_srednia") And Not SmartTags("DB_HMI_zsyp_1_dluga") Then
   			HmiRuntime.Screens("Root screen").ScreenItems("l_kr").Enabled = True
   		End If
   		If Not SmartTags("DB_HMI_zsyp_2_srednia") And Not SmartTags("DB_HMI_zsyp_2_dluga") Then
   			HmiRuntime.Screens("Root screen").ScreenItems("s_kr").Enabled = True
   		End If
   	ElseIf dlugosc_belki = "srednia" Then
   		HmiRuntime.Screens("Root screen").ScreenItems("tekst_zsyp_prawy").Text = "pnie" & Chr(10) & "-----" 
   		If Not SmartTags("DB_HMI_zsyp_1_krotka") And Not SmartTags("DB_HMI_zsyp_2_krotka") Then
   			HmiRuntime.Screens("Root screen").ScreenItems("p_kr").Enabled = True
   		End If
   		If Not SmartTags("DB_HMI_zsyp_1_dluga") And Not SmartTags("DB_HMI_zsyp_2_dluga") Then
   			HmiRuntime.Screens("Root screen").ScreenItems("p_dl").Enabled = True
   		End If
   		If Not SmartTags("DB_HMI_zsyp_1_krotka") And Not SmartTags("DB_HMI_zsyp_1_dluga") Then
   			HmiRuntime.Screens("Root screen").ScreenItems("l_sr").Enabled = True
   		End If
   		If Not SmartTags("DB_HMI_zsyp_2_krotka") And Not SmartTags("DB_HMI_zsyp_2_dluga") Then
   			HmiRuntime.Screens("Root screen").ScreenItems("s_sr").Enabled = True
   		End If
   	ElseIf dlugosc_belki = "dluga" Then
   		HmiRuntime.Screens("Root screen").ScreenItems("tekst_zsyp_prawy").Text = "pnie" & Chr(10) & "-----"
   		If Not SmartTags("DB_HMI_zsyp_1_krotka") And Not SmartTags("DB_HMI_zsyp_2_krotka") Then
   			HmiRuntime.Screens("Root screen").ScreenItems("p_kr").Enabled = True
   		End If
   		If Not SmartTags("DB_HMI_zsyp_1_srednia") And Not SmartTags("DB_HMI_zsyp_2_srednia") Then
   			HmiRuntime.Screens("Root screen").ScreenItems("p_sr").Enabled = True
   		End If
   		If Not SmartTags("DB_HMI_zsyp_1_krotka") And Not SmartTags("DB_HMI_zsyp_1_srednia") Then
   			HmiRuntime.Screens("Root screen").ScreenItems("l_dl").Enabled = True
   		End If
   		If Not SmartTags("DB_HMI_zsyp_2_krotka") And Not SmartTags("DB_HMI_zsyp_2_srednia") Then
   			HmiRuntime.Screens("Root screen").ScreenItems("s_dl").Enabled = True
   		End If 	
   	End If
   End If

VB script "Aktualizacja_nazw"
   'Skrypt służący do wyczyszczenia zapamiętanych długości belek dla danego zsypu w momencie uruchomienia trybu normalnego.
   'W przypadku uruchomienia trybu uniwersalnego odbiorcy matryca przycisków jest ukrywana oraz ustawiane są odpowiednie napisy
   'na poszczególnych zsypach
   
   If Not SmartTags("DB_HMI_odbiorca") Then	'jeżeli uruchomiono uniwersalnego odbiorcy
   	HmiRuntime.Screens("Root screen").ScreenItems("tekst_zsyp_lewy").Text = "pnie" & Chr(10) & "-----"
   	HmiRuntime.Screens("Root screen").ScreenItems("tekst_zsyp_prawy").Text = "pnie" & Chr(10) & "-----"
   	HmiRuntime.Screens("Root screen").ScreenItems("tekst_zsyp_srodkowy").Text = "Wszystkie" & Chr(10) & "pnie"
   Else	'jeżeli uruchomiono tryb normalny
   	HmiRuntime.Screens("Root screen").ScreenItems("l_kr").Enabled = True
   	HmiRuntime.Screens("Root screen").ScreenItems("l_sr").Enabled = True
   	HmiRuntime.Screens("Root screen").ScreenItems("l_dl").Enabled = True
   	HmiRuntime.Screens("Root screen").ScreenItems("p_kr").Enabled = True
   	HmiRuntime.Screens("Root screen").ScreenItems("p_sr").Enabled = True
   	HmiRuntime.Screens("Root screen").ScreenItems("p_dl").Enabled = True
   	HmiRuntime.Screens("Root screen").ScreenItems("s_kr").Enabled = True
   	HmiRuntime.Screens("Root screen").ScreenItems("s_sr").Enabled = True
   	HmiRuntime.Screens("Root screen").ScreenItems("s_dl").Enabled = True
   	SmartTags("DB_HMI_zsyp_1_krotka") = False
   	SmartTags("DB_HMI_zsyp_2_krotka") = False
   	SmartTags("DB_HMI_zsyp_3_krotka") = False
   	SmartTags("DB_HMI_zsyp_1_srednia") = False
   	SmartTags("DB_HMI_zsyp_2_srednia") = False
   	SmartTags("DB_HMI_zsyp_3_srednia") = False
   	SmartTags("DB_HMI_zsyp_1_dluga") = False
   	SmartTags("DB_HMI_zsyp_2_dluga") = False
   	SmartTags("DB_HMI_zsyp_3_dluga") = False
   	HmiRuntime.Screens("Root screen").ScreenItems("tekst_zsyp_lewy").Text = "pnie" & Chr(10) & "-----"
   	HmiRuntime.Screens("Root screen").ScreenItems("tekst_zsyp_prawy").Text = "pnie" & Chr(10) & "-----"
   	HmiRuntime.Screens("Root screen").ScreenItems("tekst_zsyp_srodkowy").Text = "pnie" & Chr(10) & "-----"
   End If
*)